Yaskawa INFORM job: apremTRJ5.JBI

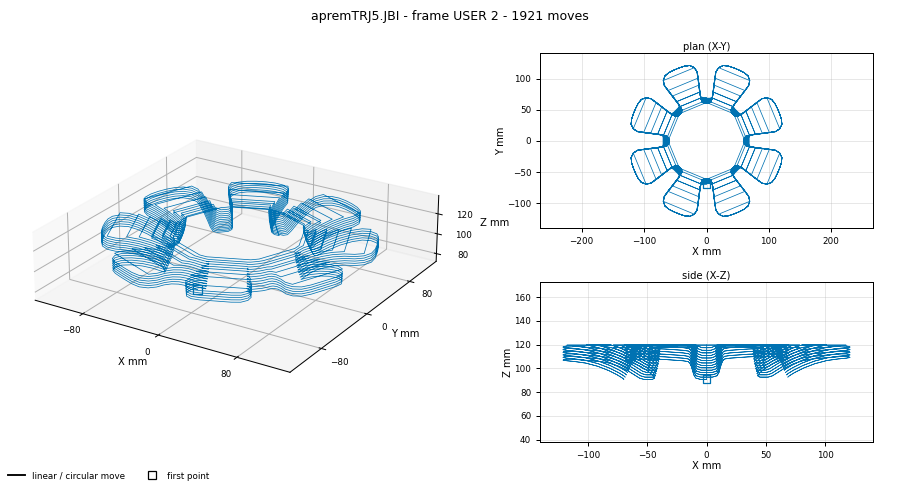
[picture p0: tool path of apremTRJ5.JBI in frame USER 2, 1921 of 1921 moves have a stored position in this frame; points joined in program order, loops and branches not executed]
/JOB
//NAME apremTRJ5
//POS
///NPOS 1921,0,0,0,0,0
///USER 2
///TOOL 1
///POSTYPE USER
///RECTAN
///RCONF 1,0,0,0,0,0,0,0,0,0,0,0,0,0,0,0,0,0,0,0,0,0,0,0
C00000=0.000,-69.663,90.662,149.0780,-0.0009,0.0000
C00001=-2.183,-69.638,90.631,149.0847,1.2932,0.0000
C00002=-5.231,-69.586,90.677,150.1957,-3.8236,0.0000
C00003=-9.064,-70.790,91.747,167.8852,-12.3668,0.0000
C00004=-10.724,-75.112,94.426,-179.6229,2.0642,0.0000
C00005=-11.710,-82.323,98.064,-179.4233,3.7476,0.0000
C00006=-12.828,-91.647,101.694,-179.3835,4.2590,0.0000
C00007=-14.066,-101.744,104.371,-179.3534,4.5111,0.0000
C00008=-15.480,-110.874,105.656,-178.6624,4.1341,0.0000
C00009=-19.937,-117.532,106.324,-177.9032,1.7507,0.0000
C00010=-26.978,-120.778,106.862,-178.7148,0.2137,0.0000
C00011=-35.142,-119.948,107.400,-179.9184,-0.0238,0.0000
C00012=-43.596,-117.150,107.753,-179.9908,-0.0034,0.0000
C00013=-52.010,-113.665,107.753,-179.9911,-0.0041,0.0000
C00014=-59.968,-109.665,107.400,-179.9255,-0.0409,0.0000
C00015=-66.327,-104.479,106.862,-179.2422,-1.0599,0.0000
C00016=-69.010,-97.206,106.324,-179.7550,-2.7196,0.0000
C00017=-67.454,-89.346,105.656,178.0185,-3.8685,0.0000
C00018=-61.998,-81.890,104.371,177.2629,-3.6488,0.0000
C00019=-55.734,-73.875,101.694,177.4206,-3.4489,0.0000
C00020=-49.931,-66.491,98.064,177.7552,-3.0586,0.0000
C00021=-45.529,-60.695,94.426,178.8066,-1.7264,0.0000
C00022=-43.647,-56.466,91.747,-179.8138,17.0577,0.0000
C00023=-45.506,-52.903,90.677,160.3117,24.3360,0.0000
C00024=-47.697,-50.786,90.631,156.2793,22.1709,0.0000
C00025=-49.259,-49.259,90.662,157.0437,22.9552,0.0000
C00026=-50.785,-47.698,90.631,157.8297,23.7213,0.0000
C00027=-52.904,-45.506,90.677,155.6631,19.6860,0.0000
C00028=-56.466,-43.647,91.747,162.9430,-0.1866,0.0000
C00029=-60.695,-45.529,94.426,-178.2736,1.1934,0.0000
C00030=-66.491,-49.931,98.064,-176.9414,2.2448,0.0000
C00031=-73.875,-55.734,101.694,-176.5511,2.5794,0.0000
C00032=-81.890,-61.998,104.371,-176.3512,2.7371,0.0000
C00033=-89.346,-67.454,105.656,-176.1315,1.9815,0.0000
C00034=-97.206,-69.010,106.324,-177.2804,-0.2450,0.0000
C00035=-104.479,-66.327,106.862,-178.9401,-0.7578,0.0000
C00036=-109.665,-59.968,107.400,-179.9591,-0.0745,0.0000
C00037=-113.665,-52.010,107.753,-179.9959,-0.0089,0.0000
C00038=-117.150,-43.596,107.753,-179.9966,-0.0092,0.0000
C00039=-119.948,-35.142,107.400,-179.9762,-0.0816,0.0000
C00040=-120.778,-26.978,106.862,179.7863,-1.2852,0.0000
C00041=-117.532,-19.937,106.324,178.2493,-2.0968,0.0000
C00042=-110.874,-15.480,105.656,175.8659,-1.3376,0.0000
C00043=-101.744,-14.066,104.371,175.4889,-0.6466,0.0000
C00044=-91.647,-12.828,101.694,175.7410,-0.6165,0.0000
C00045=-82.323,-11.710,98.064,176.2524,-0.5767,0.0000
C00046=-75.112,-10.724,94.426,177.9358,-0.3771,0.0000
C00047=-70.790,-9.064,91.747,-167.6330,12.1155,0.0000
C00048=-69.586,-5.231,90.677,-176.1790,29.8051,0.0000
C00049=-69.638,-2.184,90.631,178.7078,30.9153,0.0000
C00050=-69.663,0.000,90.662,179.9991,30.9220,0.0000
C00051=-69.638,2.183,90.631,-178.7068,30.9153,0.0000
C00052=-69.586,5.231,90.677,176.1764,29.8043,0.0000
C00053=-70.790,9.064,91.747,167.6332,12.1148,0.0000
C00054=-75.112,10.724,94.426,-177.9358,-0.3771,0.0000
C00055=-82.323,11.710,98.064,-176.2524,-0.5767,0.0000
C00056=-91.647,12.828,101.694,-175.7410,-0.6165,0.0000
C00057=-101.744,14.066,104.371,-175.4889,-0.6466,0.0000
C00058=-110.874,15.480,105.656,-175.8659,-1.3376,0.0000
C00059=-117.532,19.937,106.324,-178.2493,-2.0968,0.0000
C00060=-120.778,26.978,106.862,-179.7863,-1.2852,0.0000
C00061=-119.948,35.142,107.400,179.9762,-0.0816,0.0000
C00062=-117.150,43.596,107.753,179.9966,-0.0092,0.0000
C00063=-113.665,52.010,107.753,179.9959,-0.0089,0.0000
C00064=-109.665,59.968,107.400,179.9591,-0.0745,0.0000
C00065=-104.479,66.327,106.862,178.9401,-0.7578,0.0000
C00066=-97.206,69.010,106.324,177.2804,-0.2450,0.0000
C00067=-89.346,67.454,105.656,176.1315,1.9815,0.0000
C00068=-81.890,61.998,104.371,176.3512,2.7371,0.0000
C00069=-73.875,55.734,101.694,176.5511,2.5794,0.0000
C00070=-66.491,49.931,98.064,176.9414,2.2448,0.0000
C00071=-60.695,45.529,94.426,178.2736,1.1934,0.0000
C00072=-56.466,43.647,91.747,-162.9423,-0.1862,0.0000
C00073=-52.903,45.506,90.677,-155.6640,19.6883,0.0000
C00074=-50.786,47.697,90.631,-157.8291,23.7207,0.0000
C00075=-49.259,49.259,90.662,-157.0448,22.9563,0.0000
C00076=-47.698,50.785,90.631,-156.2787,22.1703,0.0000
C00077=-45.506,52.904,90.677,-160.3140,24.3369,0.0000
C00078=-43.647,56.466,91.747,179.8134,17.0570,0.0000
C00079=-45.529,60.695,94.426,-178.8066,-1.7264,0.0000
C00080=-49.931,66.491,98.064,-177.7552,-3.0586,0.0000
C00081=-55.734,73.875,101.694,-177.4206,-3.4489,0.0000
C00082=-61.998,81.890,104.371,-177.2629,-3.6488,0.0000
C00083=-67.454,89.346,105.656,-178.0185,-3.8685,0.0000
C00084=-69.010,97.206,106.324,179.7550,-2.7196,0.0000
C00085=-66.327,104.479,106.862,179.2422,-1.0599,0.0000
C00086=-59.968,109.665,107.400,179.9255,-0.0409,0.0000
C00087=-52.010,113.665,107.753,179.9911,-0.0041,0.0000
C00088=-43.596,117.150,107.753,179.9908,-0.0034,0.0000
C00089=-35.142,119.948,107.400,179.9184,-0.0238,0.0000
C00090=-26.978,120.778,106.862,178.7148,0.2137,0.0000
C00091=-19.937,117.532,106.324,177.9032,1.7507,0.0000
C00092=-15.480,110.874,105.656,178.6624,4.1341,0.0000
C00093=-14.066,101.744,104.371,179.3534,4.5111,0.0000
C00094=-12.828,91.647,101.694,179.3835,4.2590,0.0000
C00095=-11.710,82.323,98.064,179.4233,3.7476,0.0000
C00096=-10.724,75.112,94.426,179.6229,2.0642,0.0000
C00097=-9.064,70.790,91.747,-167.8852,-12.3668,0.0000
C00098=-5.231,69.586,90.677,-150.1957,-3.8236,0.0000
C00099=-2.183,69.638,90.631,-149.0847,1.2932,0.0000
C00100=0.000,69.663,90.662,-149.0780,-0.0009,0.0000
C00101=0.000,68.551,92.561,-150.2599,-0.0009,0.0000
C00102=2.082,68.530,92.529,-150.2645,-1.1898,0.0000
C00103=5.060,68.488,92.576,-151.4241,3.8705,0.0000
C00104=8.860,69.756,93.678,-168.9161,11.6642,0.0000
C00105=10.491,74.235,96.430,179.6271,-2.1340,0.0000
C00106=11.475,81.669,100.151,179.4707,-3.5332,0.0000
C00107=12.611,91.225,103.842,179.4509,-3.8705,0.0000
C00108=13.867,101.508,106.549,179.4410,-3.9839,0.0000
C00109=15.282,110.767,107.845,178.8532,-3.5972,0.0000
C00110=19.760,117.511,108.516,178.1979,-1.5173,0.0000
C00111=26.844,120.803,109.057,178.9013,-0.1852,0.0000
C00112=35.060,119.975,109.599,179.9308,0.0202,0.0000
C00113=43.570,117.160,109.952,179.9923,0.0029,0.0000
C00114=52.036,113.653,109.952,179.9925,0.0034,0.0000
C00115=60.044,109.627,109.599,179.9368,0.0347,0.0000
C00116=66.439,104.402,109.057,179.3540,0.9079,0.0000
C00117=69.120,97.065,108.516,179.7984,2.3465,0.0000
C00118=67.518,89.130,107.845,-178.2646,3.3542,0.0000
C00119=61.971,81.582,106.549,-177.5751,3.2135,0.0000
C00120=55.588,73.423,103.842,-177.6486,3.1262,0.0000
C00121=49.635,65.863,100.151,-177.8737,2.8734,0.0000
C00122=45.074,59.911,96.430,-178.7542,1.7728,0.0000
C00123=43.060,55.590,93.678,179.5731,-15.8809,0.0000
C00124=44.851,52.006,92.576,-161.3607,-23.4117,0.0000
C00125=46.985,49.930,92.529,-157.2861,-21.2671,0.0000
C00126=48.473,48.473,92.561,-158.0016,-21.9974,0.0000
C00127=49.930,46.986,92.529,-158.7334,-22.7144,0.0000
C00128=52.007,44.850,92.576,-156.5875,-18.6369,0.0000
C00129=55.590,43.060,93.678,-164.1198,0.4273,0.0000
C00130=59.911,45.074,96.430,178.2272,-1.2458,0.0000
C00131=65.863,49.635,100.151,177.1266,-2.1263,0.0000
C00132=73.423,55.588,103.842,176.8738,-2.3514,0.0000
C00133=81.582,61.971,106.549,176.7865,-2.4249,0.0000
C00134=89.130,67.518,107.845,176.6458,-1.7354,0.0000
C00135=97.065,69.120,108.516,177.6535,0.2016,0.0000
C00136=104.402,66.439,109.057,179.0921,0.6460,0.0000
C00137=109.627,60.044,109.599,179.9653,0.0632,0.0000
C00138=113.653,52.036,109.952,179.9966,0.0075,0.0000
C00139=117.160,43.570,109.952,179.9971,0.0077,0.0000
C00140=119.975,35.060,109.599,179.9798,0.0692,0.0000
C00141=120.803,26.844,109.057,-179.8148,1.0987,0.0000
C00142=117.511,19.760,108.516,-178.4827,1.8021,0.0000
C00143=110.767,15.282,107.845,-176.4028,1.1468,0.0000
C00144=101.508,13.867,106.549,-176.0161,0.5590,0.0000
C00145=91.225,12.611,103.842,-176.1295,0.5491,0.0000
C00146=81.669,11.475,100.151,-176.4668,0.5293,0.0000
C00147=74.235,10.491,96.430,-177.8660,0.3729,0.0000
C00148=69.756,8.860,93.678,168.3358,-11.0839,0.0000
C00149=68.488,5.060,92.576,176.1295,-28.5759,0.0000
C00150=68.530,2.082,92.529,-178.8102,-29.7355,0.0000
C00151=68.551,0.000,92.561,-179.9991,-29.7401,0.0000
C00152=68.530,-2.082,92.529,178.8093,-29.7356,0.0000
C00153=68.489,-5.060,92.576,-176.1270,-28.5749,0.0000
C00154=69.756,-8.860,93.678,-168.3360,-11.0832,0.0000
C00155=74.235,-10.491,96.430,177.8660,0.3729,0.0000
C00156=81.669,-11.475,100.151,176.4668,0.5293,0.0000
C00157=91.225,-12.611,103.842,176.1295,0.5491,0.0000
C00158=101.508,-13.867,106.549,176.0161,0.5590,0.0000
C00159=110.767,-15.282,107.845,176.4028,1.1468,0.0000
C00160=117.511,-19.760,108.516,178.4827,1.8021,0.0000
C00161=120.803,-26.844,109.057,179.8148,1.0987,0.0000
C00162=119.975,-35.060,109.599,-179.9798,0.0692,0.0000
C00163=117.160,-43.570,109.952,-179.9971,0.0077,0.0000
C00164=113.653,-52.036,109.952,-179.9966,0.0075,0.0000
C00165=109.627,-60.044,109.599,-179.9653,0.0632,0.0000
C00166=104.402,-66.439,109.057,-179.0921,0.6460,0.0000
C00167=97.065,-69.120,108.516,-177.6535,0.2016,0.0000
C00168=89.130,-67.518,107.845,-176.6458,-1.7354,0.0000
C00169=81.582,-61.971,106.549,-176.7865,-2.4249,0.0000
C00170=73.423,-55.588,103.842,-176.8738,-2.3514,0.0000
C00171=65.863,-49.635,100.151,-177.1266,-2.1263,0.0000
C00172=59.911,-45.074,96.430,-178.2272,-1.2458,0.0000
C00173=55.590,-43.060,93.678,164.1191,0.4269,0.0000
C00174=52.006,-44.851,92.576,156.5883,-18.6393,0.0000
C00175=49.930,-46.985,92.529,158.7329,-22.7139,0.0000
C00176=48.473,-48.473,92.561,158.0026,-21.9984,0.0000
C00177=46.986,-49.930,92.529,157.2856,-21.2666,0.0000
C00178=44.850,-52.007,92.576,161.3631,-23.4125,0.0000
C00179=43.060,-55.590,93.678,-179.5727,-15.8802,0.0000
C00180=45.074,-59.911,96.430,178.7542,1.7728,0.0000
C00181=49.635,-65.863,100.151,177.8737,2.8734,0.0000
C00182=55.588,-73.423,103.842,177.6486,3.1262,0.0000
C00183=61.971,-81.582,106.549,177.5751,3.2135,0.0000
C00184=67.518,-89.130,107.845,178.2646,3.3542,0.0000
C00185=69.120,-97.065,108.516,-179.7984,2.3465,0.0000
C00186=66.439,-104.402,109.057,-179.3540,0.9079,0.0000
C00187=60.044,-109.627,109.599,-179.9368,0.0347,0.0000
C00188=52.036,-113.653,109.952,-179.9925,0.0034,0.0000
C00189=43.570,-117.160,109.952,-179.9923,0.0029,0.0000
C00190=35.060,-119.975,109.599,-179.9308,0.0202,0.0000
C00191=26.844,-120.803,109.057,-178.9013,-0.1852,0.0000
C00192=19.760,-117.511,108.516,-178.1979,-1.5173,0.0000
C00193=15.282,-110.767,107.845,-178.8532,-3.5972,0.0000
C00194=13.867,-101.508,106.549,-179.4410,-3.9839,0.0000
C00195=12.611,-91.225,103.842,-179.4509,-3.8705,0.0000
C00196=11.475,-81.669,100.151,-179.4707,-3.5332,0.0000
C00197=10.491,-74.235,96.430,-179.6271,-2.1340,0.0000
C00198=8.860,-69.756,93.678,168.9161,11.6642,0.0000
C00199=5.060,-68.488,92.576,151.4241,3.8705,0.0000
C00200=2.082,-68.530,92.529,150.2645,-1.1898,0.0000
C00201=0.000,-68.551,92.561,150.2599,-0.0009,0.0000
C00202=0.000,-68.551,92.561,150.2599,-0.0009,0.0000
C00203=-2.082,-68.530,92.529,150.2644,1.1907,0.0000
C00204=-5.060,-68.489,92.576,151.4251,-3.8730,0.0000
C00205=-8.860,-69.756,93.678,168.9168,-11.6640,0.0000
C00206=-10.491,-74.235,96.430,-179.6271,2.1340,0.0000
C00207=-11.475,-81.669,100.151,-179.4707,3.5332,0.0000
C00208=-12.611,-91.225,103.842,-179.4509,3.8705,0.0000
C00209=-13.867,-101.508,106.549,-179.4410,3.9839,0.0000
C00210=-15.282,-110.767,107.845,-178.8532,3.5972,0.0000
C00211=-19.760,-117.511,108.516,-178.1979,1.5173,0.0000
C00212=-26.844,-120.803,109.057,-178.9013,0.1852,0.0000
C00213=-35.060,-119.975,109.599,-179.9308,-0.0202,0.0000
C00214=-43.570,-117.160,109.952,-179.9923,-0.0029,0.0000
C00215=-52.036,-113.653,109.952,-179.9925,-0.0034,0.0000
C00216=-60.044,-109.627,109.599,-179.9368,-0.0347,0.0000
C00217=-66.439,-104.402,109.057,-179.3540,-0.9079,0.0000
C00218=-69.120,-97.065,108.516,-179.7984,-2.3465,0.0000
C00219=-67.518,-89.130,107.845,178.2646,-3.3542,0.0000
C00220=-61.971,-81.582,106.549,177.5751,-3.2135,0.0000
C00221=-55.588,-73.423,103.842,177.6486,-3.1262,0.0000
C00222=-49.635,-65.863,100.151,177.8737,-2.8734,0.0000
C00223=-45.074,-59.911,96.430,178.7542,-1.7728,0.0000
C00224=-43.060,-55.590,93.678,-179.5731,15.8809,0.0000
C00225=-44.851,-52.006,92.576,161.3607,23.4117,0.0000
C00226=-46.985,-49.930,92.529,157.2861,21.2671,0.0000
C00227=-48.473,-48.473,92.561,158.0016,21.9974,0.0000
C00228=-49.930,-46.986,92.529,158.7334,22.7144,0.0000
C00229=-52.007,-44.850,92.576,156.5875,18.6369,0.0000
C00230=-55.590,-43.060,93.678,164.1198,-0.4273,0.0000
C00231=-59.911,-45.074,96.430,-178.2272,1.2458,0.0000
C00232=-65.863,-49.635,100.151,-177.1266,2.1263,0.0000
C00233=-73.423,-55.588,103.842,-176.8738,2.3514,0.0000
C00234=-81.582,-61.971,106.549,-176.7865,2.4249,0.0000
C00235=-89.130,-67.518,107.845,-176.6458,1.7354,0.0000
C00236=-97.065,-69.120,108.516,-177.6535,-0.2016,0.0000
C00237=-104.402,-66.439,109.057,-179.0921,-0.6460,0.0000
C00238=-109.627,-60.044,109.599,-179.9653,-0.0632,0.0000
C00239=-113.653,-52.036,109.952,-179.9966,-0.0075,0.0000
C00240=-117.160,-43.570,109.952,-179.9971,-0.0077,0.0000
C00241=-119.975,-35.060,109.599,-179.9798,-0.0692,0.0000
C00242=-120.803,-26.844,109.057,179.8148,-1.0987,0.0000
C00243=-117.511,-19.760,108.516,178.4827,-1.8021,0.0000
C00244=-110.767,-15.282,107.845,176.4028,-1.1468,0.0000
C00245=-101.508,-13.867,106.549,176.0161,-0.5590,0.0000
C00246=-91.225,-12.611,103.842,176.1295,-0.5491,0.0000
C00247=-81.669,-11.475,100.151,176.4668,-0.5293,0.0000
C00248=-74.235,-10.491,96.430,177.8660,-0.3729,0.0000
C00249=-69.756,-8.860,93.678,-168.3358,11.0839,0.0000
C00250=-68.488,-5.060,92.576,-176.1295,28.5759,0.0000
C00251=-68.530,-2.082,92.529,178.8102,29.7355,0.0000
C00252=-68.551,0.000,92.561,179.9991,29.7401,0.0000
C00253=-68.530,2.082,92.529,-178.8093,29.7356,0.0000
C00254=-68.489,5.060,92.576,176.1270,28.5749,0.0000
C00255=-69.756,8.860,93.678,168.3360,11.0832,0.0000
C00256=-74.235,10.491,96.430,-177.8660,-0.3729,0.0000
C00257=-81.669,11.475,100.151,-176.4668,-0.5293,0.0000
C00258=-91.225,12.611,103.842,-176.1295,-0.5491,0.0000
C00259=-101.508,13.867,106.549,-176.0161,-0.5590,0.0000
C00260=-110.767,15.282,107.845,-176.4028,-1.1468,0.0000
C00261=-117.511,19.760,108.516,-178.4827,-1.8021,0.0000
C00262=-120.803,26.844,109.057,-179.8148,-1.0987,0.0000
C00263=-119.975,35.060,109.599,179.9798,-0.0692,0.0000
C00264=-117.160,43.570,109.952,179.9971,-0.0077,0.0000
C00265=-113.653,52.036,109.952,179.9966,-0.0075,0.0000
C00266=-109.627,60.044,109.599,179.9653,-0.0632,0.0000
C00267=-104.402,66.439,109.057,179.0921,-0.6460,0.0000
C00268=-97.065,69.120,108.516,177.6535,-0.2016,0.0000
C00269=-89.130,67.518,107.845,176.6458,1.7354,0.0000
C00270=-81.582,61.971,106.549,176.7865,2.4249,0.0000
C00271=-73.423,55.588,103.842,176.8738,2.3514,0.0000
C00272=-65.863,49.635,100.151,177.1266,2.1263,0.0000
C00273=-59.911,45.074,96.430,178.2272,1.2458,0.0000
C00274=-55.590,43.060,93.678,-164.1191,-0.4269,0.0000
C00275=-52.006,44.851,92.576,-156.5883,18.6393,0.0000
C00276=-49.930,46.985,92.529,-158.7329,22.7139,0.0000
C00277=-48.473,48.473,92.561,-158.0026,21.9984,0.0000
C00278=-46.986,49.930,92.529,-157.2856,21.2666,0.0000
C00279=-44.850,52.007,92.576,-161.3631,23.4125,0.0000
C00280=-43.060,55.590,93.678,179.5727,15.8802,0.0000
C00281=-45.074,59.911,96.430,-178.7542,-1.7728,0.0000
C00282=-49.635,65.863,100.151,-177.8737,-2.8734,0.0000
C00283=-55.588,73.423,103.842,-177.6486,-3.1262,0.0000
C00284=-61.971,81.582,106.549,-177.5751,-3.2135,0.0000
C00285=-67.518,89.130,107.845,-178.2646,-3.3542,0.0000
C00286=-69.120,97.065,108.516,179.7984,-2.3465,0.0000
C00287=-66.439,104.402,109.057,179.3540,-0.9079,0.0000
C00288=-60.044,109.627,109.599,179.9368,-0.0347,0.0000
C00289=-52.036,113.653,109.952,179.9925,-0.0034,0.0000
C00290=-43.570,117.160,109.952,179.9923,-0.0029,0.0000
C00291=-35.060,119.975,109.599,179.9308,-0.0202,0.0000
C00292=-26.844,120.803,109.057,178.9013,0.1852,0.0000
C00293=-19.760,117.511,108.516,178.1979,1.5173,0.0000
C00294=-15.282,110.767,107.845,178.8532,3.5972,0.0000
C00295=-13.867,101.508,106.549,179.4410,3.9839,0.0000
C00296=-12.611,91.225,103.842,179.4509,3.8705,0.0000
C00297=-11.475,81.669,100.151,179.4707,3.5332,0.0000
C00298=-10.491,74.235,96.430,179.6271,2.1340,0.0000
C00299=-8.860,69.756,93.678,-168.9168,-11.6640,0.0000
C00300=-5.060,68.489,92.576,-151.4251,-3.8730,0.0000
C00301=-2.082,68.530,92.529,-150.2644,1.1907,0.0000
C00302=0.000,68.551,92.561,-150.2599,-0.0009,0.0000
C00303=0.000,67.481,94.483,-151.5573,-0.0008,0.0000
C00304=1.984,67.463,94.450,-151.5596,-1.0856,0.0000
C00305=4.895,67.432,94.499,-152.7618,3.8795,0.0000
C00306=8.665,68.764,95.632,-169.9184,10.9214,0.0000
C00307=10.271,73.406,98.456,179.6393,-2.1542,0.0000
C00308=11.257,81.064,102.255,179.5203,-3.2821,0.0000
C00309=12.417,90.845,106.000,179.5197,-3.4475,0.0000
C00310=13.694,101.302,108.733,179.5288,-3.4203,0.0000
C00311=15.114,110.675,110.036,179.0481,-3.0234,0.0000
C00312=19.611,117.493,110.711,178.5095,-1.2637,0.0000
C00313=26.731,120.823,111.254,179.1000,-0.1534,0.0000
C00314=34.993,119.997,111.797,179.9440,0.0163,0.0000
C00315=43.548,117.168,112.152,179.9938,0.0023,0.0000
C00316=52.058,113.643,112.152,179.9940,0.0028,0.0000
C00317=60.107,109.595,111.797,179.9489,0.0281,0.0000
C00318=66.533,104.337,111.254,179.4720,0.7449,0.0000
C00319=69.213,96.947,110.711,179.8395,1.9472,0.0000
C00320=67.572,88.946,110.036,-178.5336,2.8107,0.0000
C00321=61.948,81.315,108.733,-177.9127,2.7525,0.0000
C00322=55.457,73.018,106.000,-177.8999,2.7782,0.0000
C00323=49.361,65.281,102.255,-178.0167,2.6606,0.0000
C00324=44.643,59.169,98.456,-178.7313,1.7785,0.0000
C00325=42.497,54.751,95.632,179.3858,-14.6902,0.0000
C00326=44.220,51.143,94.499,-162.4610,-22.3893,0.0000
C00327=46.300,49.106,94.450,-158.3778,-20.2832,0.0000
C00328=47.716,47.716,94.483,-159.0421,-20.9569,0.0000
C00329=49.106,46.300,94.450,-159.7173,-21.6227,0.0000
C00330=51.144,44.220,94.499,-157.6099,-17.5367,0.0000
C00331=54.751,42.497,95.632,-165.3105,0.6146,0.0000
C00332=59.169,44.643,98.456,178.2215,-1.2687,0.0000
C00333=65.281,49.361,102.255,177.3394,-1.9833,0.0000
C00334=73.018,55.457,106.000,177.2218,-2.1001,0.0000
C00335=81.315,61.948,108.733,177.2475,-2.0873,0.0000
C00336=88.946,67.572,110.036,177.1893,-1.4664,0.0000
C00337=96.947,69.213,110.711,178.0528,0.1605,0.0000
C00338=104.337,66.533,111.254,179.2551,0.5280,0.0000
C00339=109.595,60.107,111.797,179.9719,0.0511,0.0000
C00340=113.643,52.058,112.152,179.9972,0.0060,0.0000
C00341=117.168,43.548,112.152,179.9977,0.0062,0.0000
C00342=119.997,34.993,111.797,179.9837,0.0560,0.0000
C00343=120.823,26.731,111.254,-179.8466,0.9000,0.0000
C00344=117.493,19.611,110.711,-178.7363,1.4905,0.0000
C00345=110.675,15.114,110.036,-176.9766,0.9519,0.0000
C00346=101.302,13.694,108.733,-176.5797,0.4712,0.0000
C00347=90.845,12.417,106.000,-176.5525,0.4803,0.0000
C00348=81.064,11.257,102.255,-176.7179,0.4797,0.0000
C00349=73.406,10.271,98.456,-177.8458,0.3607,0.0000
C00350=68.764,8.665,95.632,169.0786,-10.0816,0.0000
C00351=67.432,4.895,94.499,176.1205,-27.2382,0.0000
C00352=67.463,1.984,94.450,-178.9144,-28.4404,0.0000
C00353=67.481,0.000,94.483,-179.9992,-28.4427,0.0000
C00354=67.463,-1.984,94.450,178.9136,-28.4404,0.0000
C00355=67.432,-4.896,94.499,-176.1180,-27.2373,0.0000
C00356=68.764,-8.665,95.632,-169.0788,-10.0808,0.0000
C00357=73.406,-10.271,98.456,177.8458,0.3607,0.0000
C00358=81.064,-11.257,102.255,176.7179,0.4797,0.0000
C00359=90.845,-12.417,106.000,176.5525,0.4803,0.0000
C00360=101.302,-13.694,108.733,176.5797,0.4712,0.0000
C00361=110.675,-15.114,110.036,176.9766,0.9519,0.0000
C00362=117.493,-19.611,110.711,178.7363,1.4905,0.0000
C00363=120.823,-26.731,111.254,179.8466,0.9000,0.0000
C00364=119.997,-34.993,111.797,-179.9837,0.0560,0.0000
C00365=117.168,-43.548,112.152,-179.9977,0.0062,0.0000
C00366=113.643,-52.058,112.152,-179.9972,0.0060,0.0000
C00367=109.595,-60.107,111.797,-179.9719,0.0511,0.0000
C00368=104.337,-66.533,111.254,-179.2551,0.5280,0.0000
C00369=96.947,-69.213,110.711,-178.0528,0.1605,0.0000
C00370=88.946,-67.572,110.036,-177.1893,-1.4664,0.0000
C00371=81.315,-61.948,108.733,-177.2475,-2.0873,0.0000
C00372=73.018,-55.457,106.000,-177.2218,-2.1001,0.0000
C00373=65.281,-49.361,102.255,-177.3394,-1.9833,0.0000
C00374=59.169,-44.643,98.456,-178.2215,-1.2687,0.0000
C00375=54.751,-42.497,95.632,165.3098,0.6142,0.0000
C00376=51.143,-44.220,94.499,157.6107,-17.5390,0.0000
C00377=49.106,-46.300,94.450,159.7168,-21.6222,0.0000
C00378=47.716,-47.716,94.483,159.0431,-20.9579,0.0000
C00379=46.300,-49.106,94.450,158.3773,-20.2827,0.0000
C00380=44.220,-51.144,94.499,162.4633,-22.3901,0.0000
C00381=42.497,-54.751,95.632,-179.3854,-14.6895,0.0000
C00382=44.643,-59.169,98.456,178.7313,1.7785,0.0000
C00383=49.361,-65.281,102.255,178.0167,2.6606,0.0000
C00384=55.457,-73.018,106.000,177.8999,2.7782,0.0000
C00385=61.948,-81.315,108.733,177.9127,2.7525,0.0000
C00386=67.572,-88.946,110.036,178.5336,2.8107,0.0000
C00387=69.213,-96.947,110.711,-179.8395,1.9472,0.0000
C00388=66.533,-104.337,111.254,-179.4720,0.7449,0.0000
C00389=60.107,-109.595,111.797,-179.9489,0.0281,0.0000
C00390=52.058,-113.643,112.152,-179.9940,0.0028,0.0000
C00391=43.548,-117.168,112.152,-179.9938,0.0023,0.0000
C00392=34.993,-119.997,111.797,-179.9440,0.0163,0.0000
C00393=26.731,-120.823,111.254,-179.1000,-0.1534,0.0000
C00394=19.611,-117.493,110.711,-178.5095,-1.2637,0.0000
C00395=15.114,-110.675,110.036,-179.0481,-3.0234,0.0000
C00396=13.694,-101.302,108.733,-179.5288,-3.4203,0.0000
C00397=12.417,-90.845,106.000,-179.5197,-3.4475,0.0000
C00398=11.257,-81.064,102.255,-179.5203,-3.2821,0.0000
C00399=10.271,-73.406,98.456,-179.6393,-2.1542,0.0000
C00400=8.665,-68.764,95.632,169.9184,10.9214,0.0000
C00401=4.895,-67.432,94.499,152.7618,3.8795,0.0000
C00402=1.984,-67.463,94.450,151.5596,-1.0856,0.0000
C00403=0.000,-67.481,94.483,151.5573,-0.0008,0.0000
C00404=0.000,-67.481,94.483,151.5573,-0.0008,0.0000
C00405=-1.984,-67.463,94.450,151.5596,1.0864,0.0000
C00406=-4.896,-67.432,94.499,152.7627,-3.8820,0.0000
C00407=-8.665,-68.764,95.632,169.9192,-10.9212,0.0000
C00408=-10.271,-73.406,98.456,-179.6393,2.1542,0.0000
C00409=-11.257,-81.064,102.255,-179.5203,3.2821,0.0000
C00410=-12.417,-90.845,106.000,-179.5197,3.4475,0.0000
C00411=-13.694,-101.302,108.733,-179.5288,3.4203,0.0000
C00412=-15.114,-110.675,110.036,-179.0481,3.0234,0.0000
C00413=-19.611,-117.493,110.711,-178.5095,1.2637,0.0000
C00414=-26.731,-120.823,111.254,-179.1000,0.1534,0.0000
C00415=-34.993,-119.997,111.797,-179.9440,-0.0163,0.0000
C00416=-43.548,-117.168,112.152,-179.9938,-0.0023,0.0000
C00417=-52.058,-113.643,112.152,-179.9940,-0.0028,0.0000
C00418=-60.107,-109.595,111.797,-179.9489,-0.0281,0.0000
C00419=-66.533,-104.337,111.254,-179.4720,-0.7449,0.0000
C00420=-69.213,-96.947,110.711,-179.8395,-1.9472,0.0000
C00421=-67.572,-88.946,110.036,178.5336,-2.8107,0.0000
C00422=-61.948,-81.315,108.733,177.9127,-2.7525,0.0000
C00423=-55.457,-73.018,106.000,177.8999,-2.7782,0.0000
C00424=-49.361,-65.281,102.255,178.0167,-2.6606,0.0000
C00425=-44.643,-59.169,98.456,178.7313,-1.7785,0.0000
C00426=-42.497,-54.751,95.632,-179.3858,14.6902,0.0000
C00427=-44.220,-51.143,94.499,162.4610,22.3893,0.0000
C00428=-46.300,-49.106,94.450,158.3778,20.2832,0.0000
C00429=-47.716,-47.716,94.483,159.0421,20.9569,0.0000
C00430=-49.106,-46.300,94.450,159.7173,21.6227,0.0000
C00431=-51.144,-44.220,94.499,157.6099,17.5367,0.0000
C00432=-54.751,-42.497,95.632,165.3105,-0.6146,0.0000
C00433=-59.169,-44.643,98.456,-178.2215,1.2687,0.0000
C00434=-65.281,-49.361,102.255,-177.3394,1.9833,0.0000
C00435=-73.018,-55.457,106.000,-177.2218,2.1001,0.0000
C00436=-81.315,-61.948,108.733,-177.2475,2.0873,0.0000
C00437=-88.946,-67.572,110.036,-177.1893,1.4664,0.0000
C00438=-96.947,-69.213,110.711,-178.0528,-0.1605,0.0000
C00439=-104.337,-66.533,111.254,-179.2551,-0.5280,0.0000
C00440=-109.595,-60.107,111.797,-179.9719,-0.0511,0.0000
C00441=-113.643,-52.058,112.152,-179.9972,-0.0060,0.0000
C00442=-117.168,-43.548,112.152,-179.9977,-0.0062,0.0000
C00443=-119.997,-34.993,111.797,-179.9837,-0.0560,0.0000
C00444=-120.823,-26.731,111.254,179.8466,-0.9000,0.0000
C00445=-117.493,-19.611,110.711,178.7363,-1.4905,0.0000
C00446=-110.675,-15.114,110.036,176.9766,-0.9519,0.0000
C00447=-101.302,-13.694,108.733,176.5797,-0.4712,0.0000
C00448=-90.845,-12.417,106.000,176.5525,-0.4803,0.0000
C00449=-81.064,-11.257,102.255,176.7179,-0.4797,0.0000
C00450=-73.406,-10.271,98.456,177.8458,-0.3607,0.0000
C00451=-68.764,-8.665,95.632,-169.0786,10.0816,0.0000
C00452=-67.432,-4.895,94.499,-176.1205,27.2382,0.0000
C00453=-67.463,-1.984,94.450,178.9144,28.4404,0.0000
C00454=-67.481,0.000,94.483,179.9992,28.4427,0.0000
C00455=-67.463,1.984,94.450,-178.9136,28.4404,0.0000
C00456=-67.432,4.896,94.499,176.1180,27.2373,0.0000
C00457=-68.764,8.665,95.632,169.0788,10.0808,0.0000
C00458=-73.406,10.271,98.456,-177.8458,-0.3607,0.0000
C00459=-81.064,11.257,102.255,-176.7179,-0.4797,0.0000
C00460=-90.845,12.417,106.000,-176.5525,-0.4803,0.0000
C00461=-101.302,13.694,108.733,-176.5797,-0.4712,0.0000
C00462=-110.675,15.114,110.036,-176.9766,-0.9519,0.0000
C00463=-117.493,19.611,110.711,-178.7363,-1.4905,0.0000
C00464=-120.823,26.731,111.254,-179.8466,-0.9000,0.0000
C00465=-119.997,34.993,111.797,179.9837,-0.0560,0.0000
C00466=-117.168,43.548,112.152,179.9977,-0.0062,0.0000
C00467=-113.643,52.058,112.152,179.9972,-0.0060,0.0000
C00468=-109.595,60.107,111.797,179.9719,-0.0511,0.0000
C00469=-104.337,66.533,111.254,179.2551,-0.5280,0.0000
C00470=-96.947,69.213,110.711,178.0528,-0.1605,0.0000
C00471=-88.946,67.572,110.036,177.1893,1.4664,0.0000
C00472=-81.315,61.948,108.733,177.2475,2.0873,0.0000
C00473=-73.018,55.457,106.000,177.2218,2.1001,0.0000
C00474=-65.281,49.361,102.255,177.3394,1.9833,0.0000
C00475=-59.169,44.643,98.456,178.2215,1.2687,0.0000
C00476=-54.751,42.497,95.632,-165.3098,-0.6142,0.0000
C00477=-51.143,44.220,94.499,-157.6107,17.5390,0.0000
C00478=-49.106,46.300,94.450,-159.7168,21.6222,0.0000
C00479=-47.716,47.716,94.483,-159.0431,20.9579,0.0000
C00480=-46.300,49.106,94.450,-158.3773,20.2827,0.0000
C00481=-44.220,51.144,94.499,-162.4633,22.3901,0.0000
C00482=-42.497,54.751,95.632,179.3854,14.6895,0.0000
C00483=-44.643,59.169,98.456,-178.7313,-1.7785,0.0000
C00484=-49.361,65.281,102.255,-178.0167,-2.6606,0.0000
C00485=-55.457,73.018,106.000,-177.8999,-2.7782,0.0000
C00486=-61.948,81.315,108.733,-177.9127,-2.7525,0.0000
C00487=-67.572,88.946,110.036,-178.5336,-2.8107,0.0000
C00488=-69.213,96.947,110.711,179.8395,-1.9472,0.0000
C00489=-66.533,104.337,111.254,179.4720,-0.7449,0.0000
C00490=-60.107,109.595,111.797,179.9489,-0.0281,0.0000
C00491=-52.058,113.643,112.152,179.9940,-0.0028,0.0000
C00492=-43.548,117.168,112.152,179.9938,-0.0023,0.0000
C00493=-34.993,119.997,111.797,179.9440,-0.0163,0.0000
C00494=-26.731,120.823,111.254,179.1000,0.1534,0.0000
C00495=-19.611,117.493,110.711,178.5095,1.2637,0.0000
C00496=-15.114,110.675,110.036,179.0481,3.0234,0.0000
C00497=-13.694,101.302,108.733,179.5288,3.4203,0.0000
C00498=-12.417,90.845,106.000,179.5197,3.4475,0.0000
C00499=-11.257,81.064,102.255,179.5203,3.2821,0.0000
C00500=-10.271,73.406,98.456,179.6393,2.1542,0.0000
C00501=-8.665,68.764,95.632,-169.9192,-10.9212,0.0000
C00502=-4.896,67.432,94.499,-152.7627,-3.8820,0.0000
C00503=-1.984,67.463,94.450,-151.5596,1.0864,0.0000
C00504=0.000,67.481,94.483,-151.5573,-0.0008,0.0000
C00505=0.000,66.457,96.430,-152.9799,-0.0007,0.0000
C00506=1.891,66.441,96.396,-152.9796,-0.9804,0.0000
C00507=4.738,66.421,96.447,-154.2147,3.8448,0.0000
C00508=8.479,67.820,97.611,-170.8911,10.1417,0.0000
C00509=10.065,72.628,100.503,179.6580,-2.1261,0.0000
C00510=11.059,80.512,104.375,179.5721,-2.9949,0.0000
C00511=12.247,90.513,108.168,179.5898,-2.9910,0.0000
C00512=13.549,101.129,110.921,179.6173,-2.8213,0.0000
C00513=14.976,110.600,112.231,179.2477,-2.4139,0.0000
C00514=19.491,117.478,112.908,178.8374,-0.9912,0.0000
C00515=26.642,120.839,113.453,179.3104,-0.1186,0.0000
C00516=34.941,120.015,113.997,179.9580,0.0122,0.0000
C00517=43.531,117.175,114.352,179.9954,0.0017,0.0000
C00518=52.074,113.636,114.352,179.9956,0.0020,0.0000
C00519=60.156,109.570,113.997,179.9617,0.0211,0.0000
C00520=66.607,104.285,113.453,179.5962,0.5715,0.0000
C00521=69.288,96.852,112.908,179.8787,1.5228,0.0000
C00522=67.616,88.795,112.231,-178.8242,2.2388,0.0000
C00523=61.928,81.090,110.921,-178.2745,2.2660,0.0000
C00524=55.342,72.662,108.168,-178.1738,2.4056,0.0000
C00525=49.111,64.751,104.375,-178.1836,2.4208,0.0000
C00526=44.239,58.473,100.503,-178.7380,1.7453,0.0000
C00527=41.961,53.951,97.611,179.2487,-13.4881,0.0000
C00528=43.616,50.317,96.447,-163.6122,-21.2623,0.0000
C00529=45.644,48.318,96.396,-159.5592,-19.2137,0.0000
C00530=46.992,46.992,96.430,-160.1702,-19.8289,0.0000
C00531=48.317,45.644,96.396,-160.7867,-20.4413,0.0000
C00532=50.318,43.616,96.447,-158.7369,-16.3854,0.0000
C00533=53.952,41.961,97.611,-166.5126,0.7516,0.0000
C00534=58.473,44.239,100.503,178.2547,-1.2620,0.0000
C00535=64.751,49.111,104.375,177.5792,-1.8164,0.0000
C00536=72.662,55.342,108.168,177.5944,-1.8262,0.0000
C00537=81.090,61.928,110.921,177.7340,-1.7255,0.0000
C00538=88.795,67.616,112.231,177.7612,-1.1758,0.0000
C00539=96.852,69.288,112.908,178.4772,0.1213,0.0000
C00540=104.285,66.607,113.453,179.4285,0.4038,0.0000
C00541=109.570,60.156,113.997,179.9789,0.0383,0.0000
C00542=113.636,52.074,114.352,179.9980,0.0044,0.0000
C00543=117.175,43.531,114.352,179.9983,0.0046,0.0000
C00544=120.015,34.941,113.997,179.9878,0.0420,0.0000
C00545=120.839,26.642,113.453,-179.8814,0.6896,0.0000
C00546=117.478,19.491,112.908,-179.0088,1.1626,0.0000
C00547=110.600,14.976,112.231,-177.5861,0.7523,0.0000
C00548=101.129,13.549,110.921,-177.1787,0.3827,0.0000
C00549=90.513,12.247,108.168,-177.0090,0.4102,0.0000
C00550=80.512,11.059,104.375,-177.0051,0.4279,0.0000
C00551=72.628,10.065,100.503,-177.8739,0.3420,0.0000
C00552=67.820,8.479,97.611,169.8583,-9.1089,0.0000
C00553=66.421,4.738,96.447,176.1552,-25.7853,0.0000
C00554=66.441,1.891,96.396,-179.0196,-27.0204,0.0000
C00555=66.457,0.000,96.430,-179.9993,-27.0201,0.0000
C00556=66.441,-1.890,96.396,179.0188,-27.0205,0.0000
C00557=66.421,-4.739,96.447,-176.1528,-25.7844,0.0000
C00558=67.820,-8.479,97.611,-169.8585,-9.1082,0.0000
C00559=72.628,-10.065,100.503,177.8739,0.3420,0.0000
C00560=80.512,-11.059,104.375,177.0051,0.4279,0.0000
C00561=90.513,-12.247,108.168,177.0090,0.4102,0.0000
C00562=101.129,-13.549,110.921,177.1787,0.3827,0.0000
C00563=110.600,-14.976,112.231,177.5861,0.7523,0.0000
C00564=117.478,-19.491,112.908,179.0088,1.1626,0.0000
C00565=120.839,-26.642,113.453,179.8814,0.6896,0.0000
C00566=120.015,-34.941,113.997,-179.9878,0.0420,0.0000
C00567=117.175,-43.531,114.352,-179.9983,0.0046,0.0000
C00568=113.636,-52.074,114.352,-179.9980,0.0044,0.0000
C00569=109.570,-60.156,113.997,-179.9789,0.0383,0.0000
C00570=104.285,-66.607,113.453,-179.4285,0.4038,0.0000
C00571=96.852,-69.288,112.908,-178.4772,0.1213,0.0000
C00572=88.795,-67.616,112.231,-177.7612,-1.1758,0.0000
C00573=81.090,-61.928,110.921,-177.7340,-1.7255,0.0000
C00574=72.662,-55.342,108.168,-177.5944,-1.8262,0.0000
C00575=64.751,-49.111,104.375,-177.5792,-1.8164,0.0000
C00576=58.473,-44.239,100.503,-178.2547,-1.2620,0.0000
C00577=53.951,-41.961,97.611,166.5119,0.7513,0.0000
C00578=50.317,-43.616,96.447,158.7377,-16.3878,0.0000
C00579=48.318,-45.644,96.396,160.7863,-20.4408,0.0000
C00580=46.992,-46.992,96.430,160.1711,-19.8298,0.0000
C00581=45.644,-48.317,96.396,159.5587,-19.2133,0.0000
C00582=43.616,-50.318,96.447,163.6146,-21.2631,0.0000
C00583=41.961,-53.952,97.611,-179.2484,-13.4874,0.0000
C00584=44.239,-58.473,100.503,178.7380,1.7453,0.0000
C00585=49.111,-64.751,104.375,178.1836,2.4208,0.0000
C00586=55.342,-72.662,108.168,178.1738,2.4056,0.0000
C00587=61.928,-81.090,110.921,178.2745,2.2660,0.0000
C00588=67.616,-88.795,112.231,178.8242,2.2388,0.0000
C00589=69.288,-96.852,112.908,-179.8787,1.5228,0.0000
C00590=66.607,-104.285,113.453,-179.5962,0.5715,0.0000
C00591=60.156,-109.570,113.997,-179.9617,0.0211,0.0000
C00592=52.074,-113.636,114.352,-179.9956,0.0020,0.0000
C00593=43.531,-117.175,114.352,-179.9954,0.0017,0.0000
C00594=34.941,-120.015,113.997,-179.9580,0.0122,0.0000
C00595=26.642,-120.839,113.453,-179.3104,-0.1186,0.0000
C00596=19.491,-117.478,112.908,-178.8374,-0.9912,0.0000
C00597=14.976,-110.600,112.231,-179.2477,-2.4139,0.0000
C00598=13.549,-101.129,110.921,-179.6173,-2.8213,0.0000
C00599=12.247,-90.513,108.168,-179.5898,-2.9910,0.0000
C00600=11.059,-80.512,104.375,-179.5721,-2.9949,0.0000
C00601=10.065,-72.628,100.503,-179.6580,-2.1261,0.0000
C00602=8.479,-67.820,97.611,170.8911,10.1417,0.0000
C00603=4.738,-66.421,96.447,154.2147,3.8448,0.0000
C00604=1.891,-66.441,96.396,152.9796,-0.9804,0.0000
C00605=0.000,-66.457,96.430,152.9799,-0.0007,0.0000
C00606=0.000,-66.457,96.430,152.9799,-0.0007,0.0000
C00607=-1.890,-66.441,96.396,152.9795,0.9812,0.0000
C00608=-4.739,-66.421,96.447,154.2156,-3.8472,0.0000
C00609=-8.479,-67.820,97.611,170.8918,-10.1415,0.0000
C00610=-10.065,-72.628,100.503,-179.6580,2.1261,0.0000
C00611=-11.059,-80.512,104.375,-179.5721,2.9949,0.0000
C00612=-12.247,-90.513,108.168,-179.5898,2.9910,0.0000
C00613=-13.549,-101.129,110.921,-179.6173,2.8213,0.0000
C00614=-14.976,-110.600,112.231,-179.2477,2.4139,0.0000
C00615=-19.491,-117.478,112.908,-178.8374,0.9912,0.0000
C00616=-26.642,-120.839,113.453,-179.3104,0.1186,0.0000
C00617=-34.941,-120.015,113.997,-179.9580,-0.0122,0.0000
C00618=-43.531,-117.175,114.352,-179.9954,-0.0017,0.0000
C00619=-52.074,-113.636,114.352,-179.9956,-0.0020,0.0000
C00620=-60.156,-109.570,113.997,-179.9617,-0.0211,0.0000
C00621=-66.607,-104.285,113.453,-179.5962,-0.5715,0.0000
C00622=-69.288,-96.852,112.908,-179.8787,-1.5228,0.0000
C00623=-67.616,-88.795,112.231,178.8242,-2.2388,0.0000
C00624=-61.928,-81.090,110.921,178.2745,-2.2660,0.0000
C00625=-55.342,-72.662,108.168,178.1738,-2.4056,0.0000
C00626=-49.111,-64.751,104.375,178.1836,-2.4208,0.0000
C00627=-44.239,-58.473,100.503,178.7380,-1.7453,0.0000
C00628=-41.961,-53.951,97.611,-179.2487,13.4881,0.0000
C00629=-43.616,-50.317,96.447,163.6122,21.2623,0.0000
C00630=-45.644,-48.318,96.396,159.5592,19.2137,0.0000
C00631=-46.992,-46.992,96.430,160.1702,19.8289,0.0000
C00632=-48.317,-45.644,96.396,160.7867,20.4413,0.0000
C00633=-50.318,-43.616,96.447,158.7369,16.3854,0.0000
C00634=-53.952,-41.961,97.611,166.5126,-0.7516,0.0000
C00635=-58.473,-44.239,100.503,-178.2547,1.2620,0.0000
C00636=-64.751,-49.111,104.375,-177.5792,1.8164,0.0000
C00637=-72.662,-55.342,108.168,-177.5944,1.8262,0.0000
C00638=-81.090,-61.928,110.921,-177.7340,1.7255,0.0000
C00639=-88.795,-67.616,112.231,-177.7612,1.1758,0.0000
C00640=-96.852,-69.288,112.908,-178.4772,-0.1213,0.0000
C00641=-104.285,-66.607,113.453,-179.4285,-0.4038,0.0000
C00642=-109.570,-60.156,113.997,-179.9789,-0.0383,0.0000
C00643=-113.636,-52.074,114.352,-179.9980,-0.0044,0.0000
C00644=-117.175,-43.531,114.352,-179.9983,-0.0046,0.0000
C00645=-120.015,-34.941,113.997,-179.9878,-0.0420,0.0000
C00646=-120.839,-26.642,113.453,179.8814,-0.6896,0.0000
C00647=-117.478,-19.491,112.908,179.0088,-1.1626,0.0000
C00648=-110.600,-14.976,112.231,177.5861,-0.7523,0.0000
C00649=-101.129,-13.549,110.921,177.1787,-0.3827,0.0000
C00650=-90.513,-12.247,108.168,177.0090,-0.4102,0.0000
C00651=-80.512,-11.059,104.375,177.0051,-0.4279,0.0000
C00652=-72.628,-10.065,100.503,177.8739,-0.3420,0.0000
C00653=-67.820,-8.479,97.611,-169.8583,9.1089,0.0000
C00654=-66.421,-4.738,96.447,-176.1552,25.7853,0.0000
C00655=-66.441,-1.891,96.396,179.0196,27.0204,0.0000
C00656=-66.457,0.000,96.430,179.9993,27.0201,0.0000
C00657=-66.441,1.890,96.396,-179.0188,27.0205,0.0000
C00658=-66.421,4.739,96.447,176.1528,25.7844,0.0000
C00659=-67.820,8.479,97.611,169.8585,9.1082,0.0000
C00660=-72.628,10.065,100.503,-177.8739,-0.3420,0.0000
C00661=-80.512,11.059,104.375,-177.0051,-0.4279,0.0000
C00662=-90.513,12.247,108.168,-177.0090,-0.4102,0.0000
C00663=-101.129,13.549,110.921,-177.1787,-0.3827,0.0000
C00664=-110.600,14.976,112.231,-177.5861,-0.7523,0.0000
C00665=-117.478,19.491,112.908,-179.0088,-1.1626,0.0000
C00666=-120.839,26.642,113.453,-179.8814,-0.6896,0.0000
C00667=-120.015,34.941,113.997,179.9878,-0.0420,0.0000
C00668=-117.175,43.531,114.352,179.9983,-0.0046,0.0000
C00669=-113.636,52.074,114.352,179.9980,-0.0044,0.0000
C00670=-109.570,60.156,113.997,179.9789,-0.0383,0.0000
C00671=-104.285,66.607,113.453,179.4285,-0.4038,0.0000
C00672=-96.852,69.288,112.908,178.4772,-0.1213,0.0000
C00673=-88.795,67.616,112.231,177.7612,1.1758,0.0000
C00674=-81.090,61.928,110.921,177.7340,1.7255,0.0000
C00675=-72.662,55.342,108.168,177.5944,1.8262,0.0000
C00676=-64.751,49.111,104.375,177.5792,1.8164,0.0000
C00677=-58.473,44.239,100.503,178.2547,1.2620,0.0000
C00678=-53.951,41.961,97.611,-166.5119,-0.7513,0.0000
C00679=-50.317,43.616,96.447,-158.7377,16.3878,0.0000
C00680=-48.318,45.644,96.396,-160.7863,20.4408,0.0000
C00681=-46.992,46.992,96.430,-160.1711,19.8298,0.0000
C00682=-45.644,48.317,96.396,-159.5587,19.2133,0.0000
C00683=-43.616,50.318,96.447,-163.6146,21.2631,0.0000
C00684=-41.961,53.952,97.611,179.2484,13.4874,0.0000
C00685=-44.239,58.473,100.503,-178.7380,-1.7453,0.0000
C00686=-49.111,64.751,104.375,-178.1836,-2.4208,0.0000
C00687=-55.342,72.662,108.168,-178.1738,-2.4056,0.0000
C00688=-61.928,81.090,110.921,-178.2745,-2.2660,0.0000
C00689=-67.616,88.795,112.231,-178.8242,-2.2388,0.0000
C00690=-69.288,96.852,112.908,179.8787,-1.5228,0.0000
C00691=-66.607,104.285,113.453,179.5962,-0.5715,0.0000
C00692=-60.156,109.570,113.997,179.9617,-0.0211,0.0000
C00693=-52.074,113.636,114.352,179.9956,-0.0020,0.0000
C00694=-43.531,117.175,114.352,179.9954,-0.0017,0.0000
C00695=-34.941,120.015,113.997,179.9580,-0.0122,0.0000
C00696=-26.642,120.839,113.453,179.3104,0.1186,0.0000
C00697=-19.491,117.478,112.908,178.8374,0.9912,0.0000
C00698=-14.976,110.600,112.231,179.2477,2.4139,0.0000
C00699=-13.549,101.129,110.921,179.6173,2.8213,0.0000
C00700=-12.247,90.513,108.168,179.5898,2.9910,0.0000
C00701=-11.059,80.512,104.375,179.5721,2.9949,0.0000
C00702=-10.065,72.628,100.503,179.6580,2.1261,0.0000
C00703=-8.479,67.820,97.611,-170.8918,-10.1415,0.0000
C00704=-4.739,66.421,96.447,-154.2156,-3.8472,0.0000
C00705=-1.890,66.441,96.396,-152.9795,0.9812,0.0000
C00706=0.000,66.457,96.430,-152.9799,-0.0007,0.0000
C00707=0.000,65.484,98.403,-154.5377,-0.0007,0.0000
C00708=1.802,65.470,98.368,-154.5345,-0.8753,0.0000
C00709=4.589,65.460,98.420,-155.7900,3.7631,0.0000
C00710=8.303,66.929,99.614,-171.8345,9.3277,0.0000
C00711=9.874,71.907,102.573,179.6823,-2.0507,0.0000
C00712=10.881,80.018,106.512,179.6257,-2.6726,0.0000
C00713=12.102,90.229,110.345,179.6614,-2.5019,0.0000
C00714=13.433,100.991,113.114,179.7069,-2.1881,0.0000
C00715=14.870,110.542,114.427,179.4526,-1.7704,0.0000
C00716=19.401,117.468,115.106,179.1811,-0.7010,0.0000
C00717=26.578,120.851,115.652,179.5319,-0.0810,0.0000
C00718=34.904,120.027,116.196,179.9728,0.0079,0.0000
C00719=43.519,117.179,116.552,179.9972,0.0011,0.0000
C00720=52.086,113.631,116.552,179.9972,0.0013,0.0000
C00721=60.191,109.553,116.196,179.9752,0.0136,0.0000
C00722=66.661,104.248,115.652,179.7263,0.3883,0.0000
C00723=69.344,96.781,115.106,179.9166,1.0747,0.0000
C00724=67.651,88.679,114.427,-179.1349,1.6389,0.0000
C00725=61.913,80.909,113.114,-178.6595,1.7547,0.0000
C00726=55.244,72.359,110.345,-178.4696,2.0088,0.0000
C00727=48.887,64.275,106.512,-178.3739,2.1548,0.0000
C00728=43.864,57.827,102.573,-178.7742,1.6749,0.0000
C00729=41.455,53.197,99.614,179.1587,-12.2765,0.0000
C00730=43.043,49.532,98.420,-164.8143,-20.0240,0.0000
C00731=45.020,47.568,98.368,-160.8349,-18.0533,0.0000
C00732=46.304,46.304,98.403,-161.3911,-18.6080,0.0000
C00733=47.568,45.021,98.368,-161.9471,-19.1655,0.0000
C00734=49.533,43.042,98.420,-159.9753,-15.1834,0.0000
C00735=53.197,41.455,99.614,-167.7243,0.8416,0.0000
C00736=57.827,43.864,102.573,178.3251,-1.2258,0.0000
C00737=64.275,48.887,106.512,177.8452,-1.6261,0.0000
C00738=72.359,55.244,110.345,177.9912,-1.5304,0.0000
C00739=80.909,61.913,113.114,178.2453,-1.3405,0.0000
C00740=88.679,67.651,114.427,178.3611,-0.8651,0.0000
C00741=96.781,69.344,115.106,178.9253,0.0834,0.0000
C00742=104.248,66.661,115.652,179.6117,0.2737,0.0000
C00743=109.553,60.191,116.196,179.9864,0.0248,0.0000
C00744=113.631,52.086,116.552,179.9987,0.0028,0.0000
C00745=117.179,43.519,116.552,179.9989,0.0028,0.0000
C00746=120.027,34.904,116.196,179.9921,0.0272,0.0000
C00747=120.851,26.578,115.652,-179.9190,0.4681,0.0000
C00748=117.468,19.401,115.106,-179.2990,0.8189,0.0000
C00749=110.542,14.870,114.427,-178.2296,0.5474,0.0000
C00750=100.991,13.433,113.114,-177.8119,0.2931,0.0000
C00751=90.229,12.102,110.345,-177.4981,0.3386,0.0000
C00752=80.018,10.881,106.512,-177.3274,0.3743,0.0000
C00753=71.907,9.874,102.573,-177.9493,0.3177,0.0000
C00754=66.929,8.303,99.614,170.6723,-8.1655,0.0000
C00755=65.460,4.589,98.420,176.2369,-24.2100,0.0000
C00756=65.470,1.802,98.368,-179.1247,-25.4655,0.0000
C00757=65.484,0.000,98.403,-179.9993,-25.4623,0.0000
C00758=65.470,-1.801,98.368,179.1241,-25.4656,0.0000
C00759=65.460,-4.589,98.420,-176.2346,-24.2091,0.0000
C00760=66.929,-8.303,99.614,-170.6726,-8.1647,0.0000
C00761=71.907,-9.874,102.573,177.9493,0.3177,0.0000
C00762=80.018,-10.881,106.512,177.3274,0.3743,0.0000
C00763=90.229,-12.102,110.345,177.4981,0.3386,0.0000
C00764=100.991,-13.433,113.114,177.8119,0.2931,0.0000
C00765=110.542,-14.870,114.427,178.2296,0.5474,0.0000
C00766=117.468,-19.401,115.106,179.2990,0.8189,0.0000
C00767=120.851,-26.578,115.652,179.9190,0.4681,0.0000
C00768=120.027,-34.904,116.196,-179.9921,0.0272,0.0000
C00769=117.179,-43.519,116.552,-179.9989,0.0028,0.0000
C00770=113.631,-52.086,116.552,-179.9987,0.0028,0.0000
C00771=109.553,-60.191,116.196,-179.9864,0.0248,0.0000
C00772=104.248,-66.661,115.652,-179.6117,0.2737,0.0000
C00773=96.781,-69.344,115.106,-178.9253,0.0834,0.0000
C00774=88.679,-67.651,114.427,-178.3611,-0.8651,0.0000
C00775=80.909,-61.913,113.114,-178.2453,-1.3405,0.0000
C00776=72.359,-55.244,110.345,-177.9912,-1.5304,0.0000
C00777=64.275,-48.887,106.512,-177.8452,-1.6261,0.0000
C00778=57.827,-43.864,102.573,-178.3251,-1.2258,0.0000
C00779=53.197,-41.455,99.614,167.7235,0.8413,0.0000
C00780=49.532,-43.043,98.420,159.9760,-15.1857,0.0000
C00781=47.568,-45.020,98.368,161.9467,-19.1651,0.0000
C00782=46.304,-46.304,98.403,161.3920,-18.6089,0.0000
C00783=45.021,-47.568,98.368,160.8345,-18.0529,0.0000
C00784=43.042,-49.533,98.420,164.8166,-20.0247,0.0000
C00785=41.455,-53.197,99.614,-179.1584,-12.2757,0.0000
C00786=43.864,-57.827,102.573,178.7742,1.6749,0.0000
C00787=48.887,-64.275,106.512,178.3739,2.1548,0.0000
C00788=55.244,-72.359,110.345,178.4696,2.0088,0.0000
C00789=61.913,-80.909,113.114,178.6595,1.7547,0.0000
C00790=67.651,-88.679,114.427,179.1349,1.6389,0.0000
C00791=69.344,-96.781,115.106,-179.9166,1.0747,0.0000
C00792=66.661,-104.248,115.652,-179.7263,0.3883,0.0000
C00793=60.191,-109.553,116.196,-179.9752,0.0136,0.0000
C00794=52.086,-113.631,116.552,-179.9972,0.0013,0.0000
C00795=43.519,-117.179,116.552,-179.9972,0.0011,0.0000
C00796=34.904,-120.027,116.196,-179.9728,0.0079,0.0000
C00797=26.578,-120.851,115.652,-179.5319,-0.0810,0.0000
C00798=19.401,-117.468,115.106,-179.1811,-0.7010,0.0000
C00799=14.870,-110.542,114.427,-179.4526,-1.7704,0.0000
C00800=13.433,-100.991,113.114,-179.7069,-2.1881,0.0000
C00801=12.102,-90.229,110.345,-179.6614,-2.5019,0.0000
C00802=10.881,-80.018,106.512,-179.6257,-2.6726,0.0000
C00803=9.874,-71.907,102.573,-179.6823,-2.0507,0.0000
C00804=8.303,-66.929,99.614,171.8345,9.3277,0.0000
C00805=4.589,-65.460,98.420,155.7900,3.7631,0.0000
C00806=1.802,-65.470,98.368,154.5345,-0.8753,0.0000
C00807=0.000,-65.484,98.403,154.5377,-0.0007,0.0000
C00808=0.000,-65.484,98.403,154.5377,-0.0007,0.0000
C00809=-1.801,-65.470,98.368,154.5344,0.8759,0.0000
C00810=-4.589,-65.460,98.420,155.7909,-3.7654,0.0000
C00811=-8.303,-66.929,99.614,171.8353,-9.3274,0.0000
C00812=-9.874,-71.907,102.573,-179.6823,2.0507,0.0000
C00813=-10.881,-80.018,106.512,-179.6257,2.6726,0.0000
C00814=-12.102,-90.229,110.345,-179.6614,2.5019,0.0000
C00815=-13.433,-100.991,113.114,-179.7069,2.1881,0.0000
C00816=-14.870,-110.542,114.427,-179.4526,1.7704,0.0000
C00817=-19.401,-117.468,115.106,-179.1811,0.7010,0.0000
C00818=-26.578,-120.851,115.652,-179.5319,0.0810,0.0000
C00819=-34.904,-120.027,116.196,-179.9728,-0.0079,0.0000
C00820=-43.519,-117.179,116.552,-179.9972,-0.0011,0.0000
C00821=-52.086,-113.631,116.552,-179.9972,-0.0013,0.0000
C00822=-60.191,-109.553,116.196,-179.9752,-0.0136,0.0000
C00823=-66.661,-104.248,115.652,-179.7263,-0.3883,0.0000
C00824=-69.344,-96.781,115.106,-179.9166,-1.0747,0.0000
C00825=-67.651,-88.679,114.427,179.1349,-1.6389,0.0000
C00826=-61.913,-80.909,113.114,178.6595,-1.7547,0.0000
C00827=-55.244,-72.359,110.345,178.4696,-2.0088,0.0000
C00828=-48.887,-64.275,106.512,178.3739,-2.1548,0.0000
C00829=-43.864,-57.827,102.573,178.7742,-1.6749,0.0000
C00830=-41.455,-53.197,99.614,-179.1587,12.2765,0.0000
C00831=-43.043,-49.532,98.420,164.8143,20.0240,0.0000
C00832=-45.020,-47.568,98.368,160.8349,18.0533,0.0000
C00833=-46.304,-46.304,98.403,161.3911,18.6080,0.0000
C00834=-47.568,-45.021,98.368,161.9471,19.1655,0.0000
C00835=-49.533,-43.042,98.420,159.9753,15.1834,0.0000
C00836=-53.197,-41.455,99.614,167.7243,-0.8416,0.0000
C00837=-57.827,-43.864,102.573,-178.3251,1.2258,0.0000
C00838=-64.275,-48.887,106.512,-177.8452,1.6261,0.0000
C00839=-72.359,-55.244,110.345,-177.9912,1.5304,0.0000
C00840=-80.909,-61.913,113.114,-178.2453,1.3405,0.0000
C00841=-88.679,-67.651,114.427,-178.3611,0.8651,0.0000
C00842=-96.781,-69.344,115.106,-178.9253,-0.0834,0.0000
C00843=-104.248,-66.661,115.652,-179.6117,-0.2737,0.0000
C00844=-109.553,-60.191,116.196,-179.9864,-0.0248,0.0000
C00845=-113.631,-52.086,116.552,-179.9987,-0.0028,0.0000
C00846=-117.179,-43.519,116.552,-179.9989,-0.0028,0.0000
C00847=-120.027,-34.904,116.196,-179.9921,-0.0272,0.0000
C00848=-120.851,-26.578,115.652,179.9190,-0.4681,0.0000
C00849=-117.468,-19.401,115.106,179.2990,-0.8189,0.0000
C00850=-110.542,-14.870,114.427,178.2296,-0.5474,0.0000
C00851=-100.991,-13.433,113.114,177.8119,-0.2931,0.0000
C00852=-90.229,-12.102,110.345,177.4981,-0.3386,0.0000
C00853=-80.018,-10.881,106.512,177.3274,-0.3743,0.0000
C00854=-71.907,-9.874,102.573,177.9493,-0.3177,0.0000
C00855=-66.929,-8.303,99.614,-170.6723,8.1655,0.0000
C00856=-65.460,-4.589,98.420,-176.2369,24.2100,0.0000
C00857=-65.470,-1.802,98.368,179.1247,25.4655,0.0000
C00858=-65.484,0.000,98.403,179.9993,25.4623,0.0000
C00859=-65.470,1.801,98.368,-179.1241,25.4656,0.0000
C00860=-65.460,4.589,98.420,176.2346,24.2091,0.0000
C00861=-66.929,8.303,99.614,170.6726,8.1647,0.0000
C00862=-71.907,9.874,102.573,-177.9493,-0.3177,0.0000
C00863=-80.018,10.881,106.512,-177.3274,-0.3743,0.0000
C00864=-90.229,12.102,110.345,-177.4981,-0.3386,0.0000
C00865=-100.991,13.433,113.114,-177.8119,-0.2931,0.0000
C00866=-110.542,14.870,114.427,-178.2296,-0.5474,0.0000
C00867=-117.468,19.401,115.106,-179.2990,-0.8189,0.0000
C00868=-120.851,26.578,115.652,-179.9190,-0.4681,0.0000
C00869=-120.027,34.904,116.196,179.9921,-0.0272,0.0000
C00870=-117.179,43.519,116.552,179.9989,-0.0028,0.0000
C00871=-113.631,52.086,116.552,179.9987,-0.0028,0.0000
C00872=-109.553,60.191,116.196,179.9864,-0.0248,0.0000
C00873=-104.248,66.661,115.652,179.6117,-0.2737,0.0000
C00874=-96.781,69.344,115.106,178.9253,-0.0834,0.0000
C00875=-88.679,67.651,114.427,178.3611,0.8651,0.0000
C00876=-80.909,61.913,113.114,178.2453,1.3405,0.0000
C00877=-72.359,55.244,110.345,177.9912,1.5304,0.0000
C00878=-64.275,48.887,106.512,177.8452,1.6261,0.0000
C00879=-57.827,43.864,102.573,178.3251,1.2258,0.0000
C00880=-53.197,41.455,99.614,-167.7235,-0.8413,0.0000
C00881=-49.532,43.043,98.420,-159.9760,15.1857,0.0000
C00882=-47.568,45.020,98.368,-161.9467,19.1651,0.0000
C00883=-46.304,46.304,98.403,-161.3920,18.6089,0.0000
C00884=-45.021,47.568,98.368,-160.8345,18.0529,0.0000
C00885=-43.042,49.533,98.420,-164.8166,20.0247,0.0000
C00886=-41.455,53.197,99.614,179.1584,12.2757,0.0000
C00887=-43.864,57.827,102.573,-178.7742,-1.6749,0.0000
C00888=-48.887,64.275,106.512,-178.3739,-2.1548,0.0000
C00889=-55.244,72.359,110.345,-178.4696,-2.0088,0.0000
C00890=-61.913,80.909,113.114,-178.6595,-1.7547,0.0000
C00891=-67.651,88.679,114.427,-179.1349,-1.6389,0.0000
C00892=-69.344,96.781,115.106,179.9166,-1.0747,0.0000
C00893=-66.661,104.248,115.652,179.7263,-0.3883,0.0000
C00894=-60.191,109.553,116.196,179.9752,-0.0136,0.0000
C00895=-52.086,113.631,116.552,179.9972,-0.0013,0.0000
C00896=-43.519,117.179,116.552,179.9972,-0.0011,0.0000
C00897=-34.904,120.027,116.196,179.9728,-0.0079,0.0000
C00898=-26.578,120.851,115.652,179.5319,0.0810,0.0000
C00899=-19.401,117.468,115.106,179.1811,0.7010,0.0000
C00900=-14.870,110.542,114.427,179.4526,1.7704,0.0000
C00901=-13.433,100.991,113.114,179.7069,2.1881,0.0000
C00902=-12.102,90.229,110.345,179.6614,2.5019,0.0000
C00903=-10.881,80.018,106.512,179.6257,2.6726,0.0000
C00904=-9.874,71.907,102.573,179.6823,2.0507,0.0000
C00905=-8.303,66.929,99.614,-171.8353,-9.3274,0.0000
C00906=-4.589,65.460,98.420,-155.7909,-3.7654,0.0000
C00907=-1.801,65.470,98.368,-154.5344,0.8759,0.0000
C00908=0.000,65.484,98.403,-154.5377,-0.0007,0.0000
C00909=0.000,64.567,100.403,-156.2412,-0.0006,0.0000
C00910=1.718,64.555,100.367,-156.2347,-0.7711,0.0000
C00911=4.448,64.555,100.420,-157.4947,3.6318,0.0000
C00912=8.138,66.095,101.644,-172.7502,8.4816,0.0000
C00913=9.699,71.247,104.664,179.7112,-1.9297,0.0000
C00914=10.725,79.585,108.663,179.6813,-2.3165,0.0000
C00915=11.984,89.998,112.530,179.7347,-1.9815,0.0000
C00916=13.346,100.888,115.310,179.7980,-1.5221,0.0000
C00917=14.797,110.503,116.626,179.6633,-1.0946,0.0000
C00918=19.343,117.461,117.305,179.5402,-0.3947,0.0000
C00919=26.538,120.858,117.851,179.7639,-0.0410,0.0000
C00920=34.883,120.034,118.396,179.9883,0.0034,0.0000
C00921=43.513,117.182,118.752,179.9989,0.0004,0.0000
C00922=52.091,113.628,118.752,179.9990,0.0005,0.0000
C00923=60.210,109.543,118.396,179.9893,0.0059,0.0000
C00924=66.694,104.225,117.851,179.8621,0.1959,0.0000
C00925=69.380,96.735,117.305,179.9539,0.6042,0.0000
C00926=67.674,88.600,116.626,-179.4640,1.0121,0.0000
C00927=61.901,80.776,115.310,-179.0664,1.2192,0.0000
C00928=55.165,72.112,112.530,-178.7861,1.5888,0.0000
C00929=48.691,63.859,108.663,-178.5868,1.8636,0.0000
C00930=43.521,57.238,104.664,-178.8393,1.5689,0.0000
C00931=40.982,52.491,101.644,179.1124,-11.0563,0.0000
C00932=42.502,48.793,100.420,-166.0669,-18.6676,0.0000
C00933=44.433,46.862,100.367,-162.2097,-16.7961,0.0000
C00934=45.656,45.656,100.403,-162.7101,-17.2891,0.0000
C00935=46.862,44.433,100.367,-163.2043,-17.7906,0.0000
C00936=48.793,42.502,100.421,-161.3318,-13.9309,0.0000
C00937=52.491,40.982,101.644,-168.9445,0.8879,0.0000
C00938=57.238,43.521,104.664,178.4311,-1.1607,0.0000
C00939=63.859,48.691,108.663,178.1364,-1.4132,0.0000
C00940=72.112,55.165,112.530,178.4112,-1.2139,0.0000
C00941=80.776,61.901,115.310,178.7808,-0.9336,0.0000
C00942=88.600,67.674,116.626,178.9879,-0.5360,0.0000
C00943=96.735,69.380,117.305,179.3958,0.0461,0.0000
C00944=104.225,66.694,117.851,179.8041,0.1379,0.0000
C00945=109.543,60.210,118.396,179.9941,0.0107,0.0000
C00946=113.628,52.091,118.752,179.9995,0.0010,0.0000
C00947=117.182,43.513,118.752,179.9996,0.0011,0.0000
C00948=120.034,34.883,118.396,179.9966,0.0117,0.0000
C00949=120.858,26.538,117.851,-179.9590,0.2361,0.0000
C00950=117.461,19.343,117.305,-179.6053,0.4598,0.0000
C00951=110.503,14.797,116.626,-178.9054,0.3367,0.0000
C00952=100.888,13.346,115.310,-178.4779,0.2020,0.0000
C00953=89.998,11.984,112.530,-178.0185,0.2653,0.0000
C00954=79.585,10.725,108.663,-177.6835,0.3187,0.0000
C00955=71.247,9.699,104.664,-178.0703,0.2888,0.0000
C00956=66.095,8.138,101.644,171.5184,-7.2498,0.0000
C00957=64.555,4.448,100.420,176.3682,-22.5053,0.0000
C00958=64.555,1.718,100.367,-179.2289,-23.7653,0.0000
C00959=64.567,0.000,100.403,-179.9994,-23.7588,0.0000
C00960=64.555,-1.717,100.367,179.2283,-23.7653,0.0000
C00961=64.556,-4.448,100.421,-176.3661,-22.5043,0.0000
C00962=66.096,-8.139,101.644,-171.5187,-7.2491,0.0000
C00963=71.247,-9.699,104.664,178.0703,0.2888,0.0000
C00964=79.585,-10.725,108.663,177.6835,0.3187,0.0000
C00965=89.998,-11.984,112.530,178.0185,0.2653,0.0000
C00966=100.888,-13.346,115.310,178.4779,0.2020,0.0000
C00967=110.503,-14.797,116.626,178.9054,0.3367,0.0000
C00968=117.461,-19.343,117.305,179.6053,0.4598,0.0000
C00969=120.858,-26.538,117.851,179.9590,0.2361,0.0000
C00970=120.034,-34.883,118.396,-179.9966,0.0117,0.0000
C00971=117.182,-43.513,118.752,-179.9996,0.0011,0.0000
C00972=113.628,-52.091,118.752,-179.9995,0.0010,0.0000
C00973=109.543,-60.210,118.396,-179.9941,0.0107,0.0000
C00974=104.225,-66.694,117.851,-179.8041,0.1379,0.0000
C00975=96.735,-69.380,117.305,-179.3958,0.0461,0.0000
C00976=88.600,-67.674,116.626,-178.9879,-0.5360,0.0000
C00977=80.776,-61.901,115.310,-178.7808,-0.9336,0.0000
C00978=72.112,-55.165,112.530,-178.4112,-1.2139,0.0000
C00979=63.859,-48.691,108.663,-178.1364,-1.4132,0.0000
C00980=57.238,-43.521,104.664,-178.4311,-1.1607,0.0000
C00981=52.491,-40.982,101.644,168.9437,0.8876,0.0000
C00982=48.793,-42.502,100.420,161.3324,-13.9331,0.0000
C00983=46.862,-44.433,100.367,163.2039,-17.7903,0.0000
C00984=45.656,-45.656,100.403,162.7109,-17.2899,0.0000
C00985=44.433,-46.862,100.367,162.2094,-16.7957,0.0000
C00986=42.502,-48.793,100.421,166.0691,-18.6682,0.0000
C00987=40.982,-52.491,101.644,-179.1121,-11.0555,0.0000
C00988=43.521,-57.238,104.664,178.8393,1.5689,0.0000
C00989=48.691,-63.859,108.663,178.5868,1.8636,0.0000
C00990=55.165,-72.112,112.530,178.7861,1.5888,0.0000
C00991=61.901,-80.776,115.310,179.0664,1.2192,0.0000
C00992=67.674,-88.600,116.626,179.4640,1.0121,0.0000
C00993=69.380,-96.735,117.305,-179.9539,0.6042,0.0000
C00994=66.694,-104.225,117.851,-179.8621,0.1959,0.0000
C00995=60.210,-109.543,118.396,-179.9893,0.0059,0.0000
C00996=52.091,-113.628,118.752,-179.9990,0.0005,0.0000
C00997=43.513,-117.182,118.752,-179.9989,0.0004,0.0000
C00998=34.883,-120.034,118.396,-179.9883,0.0034,0.0000
C00999=26.538,-120.858,117.851,-179.7639,-0.0410,0.0000
C01000=19.343,-117.461,117.305,-179.5402,-0.3947,0.0000
C01001=14.797,-110.503,116.626,-179.6633,-1.0946,0.0000
C01002=13.346,-100.888,115.310,-179.7980,-1.5221,0.0000
C01003=11.984,-89.998,112.530,-179.7347,-1.9815,0.0000
C01004=10.725,-79.585,108.663,-179.6813,-2.3165,0.0000
C01005=9.699,-71.247,104.664,-179.7112,-1.9297,0.0000
C01006=8.138,-66.095,101.644,172.7502,8.4816,0.0000
C01007=4.448,-64.555,100.420,157.4947,3.6318,0.0000
C01008=1.718,-64.555,100.367,156.2347,-0.7711,0.0000
C01009=0.000,-64.567,100.403,156.2412,-0.0006,0.0000
C01010=0.000,-64.567,100.403,156.2412,-0.0006,0.0000
C01011=-1.717,-64.555,100.367,156.2347,0.7717,0.0000
C01012=-4.448,-64.556,100.421,157.4957,-3.6339,0.0000
C01013=-8.139,-66.096,101.644,172.7509,-8.4813,0.0000
C01014=-9.699,-71.247,104.664,-179.7112,1.9297,0.0000
C01015=-10.725,-79.585,108.663,-179.6813,2.3165,0.0000
C01016=-11.984,-89.998,112.530,-179.7347,1.9815,0.0000
C01017=-13.346,-100.888,115.310,-179.7980,1.5221,0.0000
C01018=-14.797,-110.503,116.626,-179.6633,1.0946,0.0000
C01019=-19.343,-117.461,117.305,-179.5402,0.3947,0.0000
C01020=-26.538,-120.858,117.851,-179.7639,0.0410,0.0000
C01021=-34.883,-120.034,118.396,-179.9883,-0.0034,0.0000
C01022=-43.513,-117.182,118.752,-179.9989,-0.0004,0.0000
C01023=-52.091,-113.628,118.752,-179.9990,-0.0005,0.0000
C01024=-60.210,-109.543,118.396,-179.9893,-0.0059,0.0000
C01025=-66.694,-104.225,117.851,-179.8621,-0.1959,0.0000
C01026=-69.380,-96.735,117.305,-179.9539,-0.6042,0.0000
C01027=-67.674,-88.600,116.626,179.4640,-1.0121,0.0000
C01028=-61.901,-80.776,115.310,179.0664,-1.2192,0.0000
C01029=-55.165,-72.112,112.530,178.7861,-1.5888,0.0000
C01030=-48.691,-63.859,108.663,178.5868,-1.8636,0.0000
C01031=-43.521,-57.238,104.664,178.8393,-1.5689,0.0000
C01032=-40.982,-52.491,101.644,-179.1124,11.0563,0.0000
C01033=-42.502,-48.793,100.420,166.0669,18.6676,0.0000
C01034=-44.433,-46.862,100.367,162.2097,16.7961,0.0000
C01035=-45.656,-45.656,100.403,162.7101,17.2891,0.0000
C01036=-46.862,-44.433,100.367,163.2043,17.7906,0.0000
C01037=-48.793,-42.502,100.421,161.3318,13.9309,0.0000
C01038=-52.491,-40.982,101.644,168.9445,-0.8879,0.0000
C01039=-57.238,-43.521,104.664,-178.4311,1.1607,0.0000
C01040=-63.859,-48.691,108.663,-178.1364,1.4132,0.0000
C01041=-72.112,-55.165,112.530,-178.4112,1.2139,0.0000
C01042=-80.776,-61.901,115.310,-178.7808,0.9336,0.0000
C01043=-88.600,-67.674,116.626,-178.9879,0.5360,0.0000
C01044=-96.735,-69.380,117.305,-179.3958,-0.0461,0.0000
C01045=-104.225,-66.694,117.851,-179.8041,-0.1379,0.0000
C01046=-109.543,-60.210,118.396,-179.9941,-0.0107,0.0000
C01047=-113.628,-52.091,118.752,-179.9995,-0.0010,0.0000
C01048=-117.182,-43.513,118.752,-179.9996,-0.0011,0.0000
C01049=-120.034,-34.883,118.396,-179.9966,-0.0117,0.0000
C01050=-120.858,-26.538,117.851,179.9590,-0.2361,0.0000
C01051=-117.461,-19.343,117.305,179.6053,-0.4598,0.0000
C01052=-110.503,-14.797,116.626,178.9054,-0.3367,0.0000
C01053=-100.888,-13.346,115.310,178.4779,-0.2020,0.0000
C01054=-89.998,-11.984,112.530,178.0185,-0.2653,0.0000
C01055=-79.585,-10.725,108.663,177.6835,-0.3187,0.0000
C01056=-71.247,-9.699,104.664,178.0703,-0.2888,0.0000
C01057=-66.095,-8.138,101.644,-171.5184,7.2498,0.0000
C01058=-64.555,-4.448,100.420,-176.3682,22.5053,0.0000
C01059=-64.555,-1.718,100.367,179.2289,23.7653,0.0000
C01060=-64.567,0.000,100.403,179.9994,23.7588,0.0000
C01061=-64.555,1.717,100.367,-179.2283,23.7653,0.0000
C01062=-64.556,4.448,100.421,176.3661,22.5043,0.0000
C01063=-66.096,8.139,101.644,171.5187,7.2491,0.0000
C01064=-71.247,9.699,104.664,-178.0703,-0.2888,0.0000
C01065=-79.585,10.725,108.663,-177.6835,-0.3187,0.0000
C01066=-89.998,11.984,112.530,-178.0185,-0.2653,0.0000
C01067=-100.888,13.346,115.310,-178.4779,-0.2020,0.0000
C01068=-110.503,14.797,116.626,-178.9054,-0.3367,0.0000
C01069=-117.461,19.343,117.305,-179.6053,-0.4598,0.0000
C01070=-120.858,26.538,117.851,-179.9590,-0.2361,0.0000
C01071=-120.034,34.883,118.396,179.9966,-0.0117,0.0000
C01072=-117.182,43.513,118.752,179.9996,-0.0011,0.0000
C01073=-113.628,52.091,118.752,179.9995,-0.0010,0.0000
C01074=-109.543,60.210,118.396,179.9941,-0.0107,0.0000
C01075=-104.225,66.694,117.851,179.8041,-0.1379,0.0000
C01076=-96.735,69.380,117.305,179.3958,-0.0461,0.0000
C01077=-88.600,67.674,116.626,178.9879,0.5360,0.0000
C01078=-80.776,61.901,115.310,178.7808,0.9336,0.0000
C01079=-72.112,55.165,112.530,178.4112,1.2139,0.0000
C01080=-63.859,48.691,108.663,178.1364,1.4132,0.0000
C01081=-57.238,43.521,104.664,178.4311,1.1607,0.0000
C01082=-52.491,40.982,101.644,-168.9437,-0.8876,0.0000
C01083=-48.793,42.502,100.420,-161.3324,13.9331,0.0000
C01084=-46.862,44.433,100.367,-163.2039,17.7903,0.0000
C01085=-45.656,45.656,100.403,-162.7109,17.2899,0.0000
C01086=-44.433,46.862,100.367,-162.2094,16.7957,0.0000
C01087=-42.502,48.793,100.421,-166.0691,18.6682,0.0000
C01088=-40.982,52.491,101.644,179.1121,11.0555,0.0000
C01089=-43.521,57.238,104.664,-178.8393,-1.5689,0.0000
C01090=-48.691,63.859,108.663,-178.5868,-1.8636,0.0000
C01091=-55.165,72.112,112.530,-178.7861,-1.5888,0.0000
C01092=-61.901,80.776,115.310,-179.0664,-1.2192,0.0000
C01093=-67.674,88.600,116.626,-179.4640,-1.0121,0.0000
C01094=-69.380,96.735,117.305,179.9539,-0.6042,0.0000
C01095=-66.694,104.225,117.851,179.8621,-0.1959,0.0000
C01096=-60.210,109.543,118.396,179.9893,-0.0059,0.0000
C01097=-52.091,113.628,118.752,179.9990,-0.0005,0.0000
C01098=-43.513,117.182,118.752,179.9989,-0.0004,0.0000
C01099=-34.883,120.034,118.396,179.9883,-0.0034,0.0000
C01100=-26.538,120.858,117.851,179.7639,0.0410,0.0000
C01101=-19.343,117.461,117.305,179.5402,0.3947,0.0000
C01102=-14.797,110.503,116.626,179.6633,1.0946,0.0000
C01103=-13.346,100.888,115.310,179.7980,1.5221,0.0000
C01104=-11.984,89.998,112.530,179.7347,1.9815,0.0000
C01105=-10.725,79.585,108.663,179.6813,2.3165,0.0000
C01106=-9.699,71.247,104.664,179.7112,1.9297,0.0000
C01107=-8.139,66.096,101.644,-172.7509,-8.4813,0.0000
C01108=-4.448,64.556,100.421,-157.4957,-3.6339,0.0000
C01109=-1.717,64.555,100.367,-156.2347,0.7717,0.0000
C01110=0.000,64.567,100.403,-156.2412,-0.0006,0.0000
C01111=0.000,63.713,102.430,-158.1009,-0.0005,0.0000
C01112=1.640,63.703,102.394,-158.0906,-0.6691,0.0000
C01113=4.317,63.713,102.448,-159.3359,3.4482,0.0000
C01114=7.987,65.326,103.699,-173.6400,7.6051,0.0000
C01115=9.542,70.656,106.778,179.7440,-1.7650,0.0000
C01116=10.593,79.218,110.828,179.7386,-1.9280,0.0000
C01117=11.894,89.822,114.721,179.8100,-1.4313,0.0000
C01118=13.292,100.823,117.508,179.8911,-0.8249,0.0000
C01119=14.760,110.482,118.825,179.8808,-0.3886,0.0000
C01120=19.318,117.458,119.505,179.9140,-0.0739,0.0000
C01121=69.395,96.715,119.505,179.9914,0.1131,0.0000
C01122=67.686,88.559,118.825,-179.8095,0.3590,0.0000
C01123=61.894,80.692,117.508,-179.4936,0.6603,0.0000
C01124=55.104,71.924,114.721,-179.1222,1.1465,0.0000
C01125=48.525,63.506,110.828,-178.8212,1.5483,0.0000
C01126=43.214,56.709,106.778,-178.9327,1.4292,0.0000
C01127=40.545,51.840,103.699,179.1064,-9.8277,0.0000
C01128=41.999,48.104,102.448,-167.3698,-17.1865,0.0000
C01129=43.885,46.204,102.394,-163.6880,-15.4365,0.0000
C01130=45.052,45.052,102.430,-164.1323,-15.8671,0.0000
C01131=46.204,43.886,102.394,-164.5638,-16.3122,0.0000
C01132=48.104,41.999,102.448,-162.8129,-12.6281,0.0000
C01133=51.840,40.545,103.699,-170.1730,0.8939,0.0000
C01134=56.709,43.214,106.778,178.5708,-1.0673,0.0000
C01135=63.506,48.525,110.828,178.4517,-1.1788,0.0000
C01136=71.924,55.104,114.721,178.8535,-0.8778,0.0000
C01137=80.692,61.894,117.508,179.3397,-0.5064,0.0000
C01138=88.559,67.686,118.825,179.6410,-0.1905,0.0000
C01139=96.715,69.395,119.505,179.8869,0.0086,0.0000
C01140=117.458,19.318,119.505,-179.9261,0.0860,0.0000
C01141=110.482,14.760,118.825,-179.6114,0.1192,0.0000
C01142=100.823,13.292,117.508,-179.1751,0.1089,0.0000
C01143=89.822,11.894,114.721,-178.5687,0.1900,0.0000
C01144=79.218,10.593,110.828,-178.0720,0.2614,0.0000
C01145=70.656,9.542,106.778,-178.2350,0.2560,0.0000
C01146=65.326,7.987,103.699,172.3949,-6.3600,0.0000
C01147=63.713,4.317,102.448,176.5518,-20.6641,0.0000
C01148=63.703,1.640,102.394,-179.3309,-21.9094,0.0000
C01149=63.713,0.000,102.430,-179.9995,-21.8991,0.0000
C01150=63.703,-1.639,102.394,179.3305,-21.9094,0.0000
C01151=63.713,-4.317,102.448,-176.5498,-20.6631,0.0000
C01152=65.326,-7.987,103.699,-172.3952,-6.3593,0.0000
C01153=70.656,-9.542,106.778,178.2350,0.2560,0.0000
C01154=79.218,-10.593,110.828,178.0720,0.2614,0.0000
C01155=89.822,-11.894,114.721,178.5687,0.1900,0.0000
C01156=100.823,-13.292,117.508,179.1751,0.1089,0.0000
C01157=110.482,-14.760,118.825,179.6114,0.1192,0.0000
C01158=117.458,-19.318,119.505,179.9261,0.0860,0.0000
C01159=96.715,-69.395,119.505,-179.8869,0.0086,0.0000
C01160=88.559,-67.686,118.825,-179.6410,-0.1905,0.0000
C01161=80.692,-61.894,117.508,-179.3397,-0.5064,0.0000
C01162=71.924,-55.104,114.721,-178.8535,-0.8778,0.0000
C01163=63.506,-48.525,110.828,-178.4517,-1.1788,0.0000
C01164=56.709,-43.214,106.778,-178.5708,-1.0673,0.0000
C01165=51.840,-40.545,103.699,170.1723,0.8936,0.0000
C01166=48.104,-41.999,102.448,162.8135,-12.6302,0.0000
C01167=46.204,-43.885,102.394,164.5635,-16.3120,0.0000
C01168=45.052,-45.052,102.430,164.1329,-15.8677,0.0000
C01169=43.886,-46.204,102.394,163.6878,-15.4362,0.0000
C01170=41.999,-48.104,102.448,167.3719,-17.1871,0.0000
C01171=40.545,-51.840,103.699,-179.1061,-9.8270,0.0000
C01172=43.214,-56.709,106.778,178.9327,1.4292,0.0000
C01173=48.525,-63.506,110.828,178.8212,1.5483,0.0000
C01174=55.104,-71.924,114.721,179.1222,1.1465,0.0000
C01175=61.894,-80.692,117.508,179.4936,0.6603,0.0000
C01176=67.686,-88.559,118.825,179.8095,0.3590,0.0000
C01177=69.395,-96.715,119.505,-179.9914,0.1131,0.0000
C01178=19.318,-117.458,119.505,-179.9140,-0.0739,0.0000
C01179=14.760,-110.482,118.825,-179.8808,-0.3886,0.0000
C01180=13.292,-100.823,117.508,-179.8911,-0.8249,0.0000
C01181=11.894,-89.822,114.721,-179.8100,-1.4313,0.0000
C01182=10.593,-79.218,110.828,-179.7386,-1.9280,0.0000
C01183=9.542,-70.656,106.778,-179.7440,-1.7650,0.0000
C01184=7.987,-65.326,103.699,173.6400,7.6051,0.0000
C01185=4.317,-63.713,102.448,159.3359,3.4482,0.0000
C01186=1.640,-63.703,102.394,158.0906,-0.6691,0.0000
C01187=0.000,-63.713,102.430,158.1009,-0.0005,0.0000
C01188=0.000,-63.713,102.430,158.1009,-0.0005,0.0000
C01189=-1.639,-63.703,102.394,158.0906,0.6695,0.0000
C01190=-4.317,-63.713,102.448,159.3369,-3.4502,0.0000
C01191=-7.987,-65.326,103.699,173.6407,-7.6048,0.0000
C01192=-9.542,-70.656,106.778,-179.7440,1.7650,0.0000
C01193=-10.593,-79.218,110.828,-179.7386,1.9280,0.0000
C01194=-11.894,-89.822,114.721,-179.8100,1.4313,0.0000
C01195=-13.292,-100.823,117.508,-179.8911,0.8249,0.0000
C01196=-14.760,-110.482,118.825,-179.8808,0.3886,0.0000
C01197=-19.318,-117.458,119.505,-179.9140,0.0739,0.0000
C01198=-69.395,-96.715,119.505,-179.9914,-0.1131,0.0000
C01199=-67.686,-88.559,118.825,179.8095,-0.3590,0.0000
C01200=-61.894,-80.692,117.508,179.4936,-0.6603,0.0000
C01201=-55.104,-71.924,114.721,179.1222,-1.1465,0.0000
C01202=-48.525,-63.506,110.828,178.8212,-1.5483,0.0000
C01203=-43.214,-56.709,106.778,178.9327,-1.4292,0.0000
C01204=-40.545,-51.840,103.699,-179.1064,9.8277,0.0000
C01205=-41.999,-48.104,102.448,167.3698,17.1865,0.0000
C01206=-43.885,-46.204,102.394,163.6880,15.4365,0.0000
C01207=-45.052,-45.052,102.430,164.1323,15.8671,0.0000
C01208=-46.204,-43.886,102.394,164.5638,16.3122,0.0000
C01209=-48.104,-41.999,102.448,162.8129,12.6281,0.0000
C01210=-51.840,-40.545,103.699,170.1730,-0.8939,0.0000
C01211=-56.709,-43.214,106.778,-178.5708,1.0673,0.0000
C01212=-63.506,-48.525,110.828,-178.4517,1.1788,0.0000
C01213=-71.924,-55.104,114.721,-178.8535,0.8778,0.0000
C01214=-80.692,-61.894,117.508,-179.3397,0.5064,0.0000
C01215=-88.559,-67.686,118.825,-179.6410,0.1905,0.0000
C01216=-96.715,-69.395,119.505,-179.8869,-0.0086,0.0000
C01217=-117.458,-19.318,119.505,179.9261,-0.0860,0.0000
C01218=-110.482,-14.760,118.825,179.6114,-0.1192,0.0000
C01219=-100.823,-13.292,117.508,179.1751,-0.1089,0.0000
C01220=-89.822,-11.894,114.721,178.5687,-0.1900,0.0000
C01221=-79.218,-10.593,110.828,178.0720,-0.2614,0.0000
C01222=-70.656,-9.542,106.778,178.2350,-0.2560,0.0000
C01223=-65.326,-7.987,103.699,-172.3949,6.3600,0.0000
C01224=-63.713,-4.317,102.448,-176.5518,20.6641,0.0000
C01225=-63.703,-1.640,102.394,179.3309,21.9094,0.0000
C01226=-63.713,0.000,102.430,179.9995,21.8991,0.0000
C01227=-63.703,1.639,102.394,-179.3305,21.9094,0.0000
C01228=-63.713,4.317,102.448,176.5498,20.6631,0.0000
C01229=-65.326,7.987,103.699,172.3952,6.3593,0.0000
C01230=-70.656,9.542,106.778,-178.2350,-0.2560,0.0000
C01231=-79.218,10.593,110.828,-178.0720,-0.2614,0.0000
C01232=-89.822,11.894,114.721,-178.5687,-0.1900,0.0000
C01233=-100.823,13.292,117.508,-179.1751,-0.1089,0.0000
C01234=-110.482,14.760,118.825,-179.6114,-0.1192,0.0000
C01235=-117.458,19.318,119.505,-179.9261,-0.0860,0.0000
C01236=-96.715,69.395,119.505,179.8869,-0.0086,0.0000
C01237=-88.559,67.686,118.825,179.6410,0.1905,0.0000
C01238=-80.692,61.894,117.508,179.3397,0.5064,0.0000
C01239=-71.924,55.104,114.721,178.8535,0.8778,0.0000
C01240=-63.506,48.525,110.828,178.4517,1.1788,0.0000
C01241=-56.709,43.214,106.778,178.5708,1.0673,0.0000
C01242=-51.840,40.545,103.699,-170.1723,-0.8936,0.0000
C01243=-48.104,41.999,102.448,-162.8135,12.6302,0.0000
C01244=-46.204,43.885,102.394,-164.5635,16.3120,0.0000
C01245=-45.052,45.052,102.430,-164.1329,15.8677,0.0000
C01246=-43.886,46.204,102.394,-163.6878,15.4362,0.0000
C01247=-41.999,48.104,102.448,-167.3719,17.1871,0.0000
C01248=-40.545,51.840,103.699,179.1061,9.8270,0.0000
C01249=-43.214,56.709,106.778,-178.9327,-1.4292,0.0000
C01250=-48.525,63.506,110.828,-178.8212,-1.5483,0.0000
C01251=-55.104,71.924,114.721,-179.1222,-1.1465,0.0000
C01252=-61.894,80.692,117.508,-179.4936,-0.6603,0.0000
C01253=-67.686,88.559,118.825,-179.8095,-0.3590,0.0000
C01254=-69.395,96.715,119.505,179.9914,-0.1131,0.0000
C01255=-19.318,117.458,119.505,179.9140,0.0739,0.0000
C01256=-14.760,110.482,118.825,179.8808,0.3886,0.0000
C01257=-13.292,100.823,117.508,179.8911,0.8249,0.0000
C01258=-11.894,89.822,114.721,179.8100,1.4313,0.0000
C01259=-10.593,79.218,110.828,179.7386,1.9280,0.0000
C01260=-9.542,70.656,106.778,179.7440,1.7650,0.0000
C01261=-7.987,65.326,103.699,-173.6407,-7.6048,0.0000
C01262=-4.317,63.713,102.448,-159.3369,-3.4502,0.0000
C01263=-1.639,63.703,102.394,-158.0906,0.6695,0.0000
C01264=0.000,63.713,102.430,-158.1009,-0.0005,0.0000
C01265=0.000,62.929,104.486,-160.1268,-0.0004,0.0000
C01266=1.568,62.919,104.448,-160.1124,-0.5703,0.0000
C01267=4.196,62.938,104.504,-161.3200,3.2108,0.0000
C01268=7.849,64.627,105.781,-174.5070,6.6994,0.0000
C01269=9.405,70.138,108.911,179.7800,-1.5589,0.0000
C01270=10.487,78.922,113.006,179.7979,-1.5091,0.0000
C01271=11.833,89.705,116.917,179.8874,-0.8532,0.0000
C01272=13.270,100.797,119.708,179.9870,-0.0985,0.0000
C01273=61.891,80.658,119.708,-179.9395,0.0788,0.0000
C01274=55.063,71.798,116.917,-179.4764,0.6829,0.0000
C01275=48.391,63.222,113.006,-179.0757,1.2101,0.0000
C01276=42.945,56.245,108.911,-179.0531,1.2579,0.0000
C01277=40.148,51.249,105.781,179.1373,-8.5900,0.0000
C01278=41.537,47.471,104.504,-168.7231,-15.5750,0.0000
C01279=43.382,45.599,104.448,-165.2737,-13.9692,0.0000
C01280=44.497,44.497,104.486,-165.6622,-14.3373,0.0000
C01281=45.599,43.382,104.448,-166.0310,-14.7265,0.0000
C01282=47.472,41.536,104.504,-164.4245,-11.2750,0.0000
C01283=51.249,40.149,105.781,-171.4107,0.8630,0.0000
C01284=56.245,42.945,108.911,178.7421,-0.9469,0.0000
C01285=63.222,48.391,113.006,178.7899,-0.9243,0.0000
C01286=71.798,55.063,116.917,179.3171,-0.5236,0.0000
C01287=80.658,61.891,119.708,179.9212,-0.0605,0.0000
C01288=100.797,13.270,119.708,-179.9015,0.0130,0.0000
C01289=89.705,11.833,116.917,-179.1468,0.1126,0.0000
C01290=78.922,10.487,113.006,-178.4909,0.2021,0.0000
C01291=70.138,9.405,108.911,-178.4411,0.2200,0.0000
C01292=64.627,7.849,105.781,173.3006,-5.4930,0.0000
C01293=62.938,4.196,104.504,176.7892,-18.6800,0.0000
C01294=62.919,1.568,104.448,-179.4297,-19.8876,0.0000
C01295=62.929,0.000,104.486,-179.9996,-19.8732,0.0000
C01296=62.919,-1.567,104.448,179.4294,-19.8876,0.0000
C01297=62.938,-4.197,104.504,-176.7874,-18.6791,0.0000
C01298=64.628,-7.849,105.781,-173.3009,-5.4923,0.0000
C01299=70.138,-9.405,108.911,178.4411,0.2200,0.0000
C01300=78.922,-10.487,113.006,178.4909,0.2021,0.0000
C01301=89.705,-11.833,116.917,179.1468,0.1126,0.0000
C01302=100.797,-13.270,119.708,179.9015,0.0130,0.0000
C01303=80.658,-61.891,119.708,-179.9212,-0.0605,0.0000
C01304=71.798,-55.063,116.917,-179.3171,-0.5236,0.0000
C01305=63.222,-48.391,113.006,-178.7899,-0.9243,0.0000
C01306=56.245,-42.945,108.911,-178.7421,-0.9469,0.0000
C01307=51.249,-40.148,105.781,171.4100,0.8627,0.0000
C01308=47.471,-41.537,104.504,164.4250,-11.2769,0.0000
C01309=45.599,-43.382,104.448,166.0308,-14.7263,0.0000
C01310=44.497,-44.497,104.486,165.6627,-14.3378,0.0000
C01311=43.382,-45.599,104.448,165.2735,-13.9690,0.0000
C01312=41.536,-47.472,104.504,168.7250,-15.5755,0.0000
C01313=40.149,-51.249,105.781,-179.1370,-8.5893,0.0000
C01314=42.945,-56.245,108.911,179.0531,1.2579,0.0000
C01315=48.391,-63.222,113.006,179.0757,1.2101,0.0000
C01316=55.063,-71.798,116.917,179.4764,0.6829,0.0000
C01317=61.891,-80.658,119.708,179.9395,0.0788,0.0000
C01318=13.270,-100.797,119.708,-179.9870,-0.0985,0.0000
C01319=11.833,-89.705,116.917,-179.8874,-0.8532,0.0000
C01320=10.487,-78.922,113.006,-179.7979,-1.5091,0.0000
C01321=9.405,-70.138,108.911,-179.7800,-1.5589,0.0000
C01322=7.849,-64.627,105.781,174.5070,6.6994,0.0000
C01323=4.196,-62.938,104.504,161.3200,3.2108,0.0000
C01324=1.568,-62.919,104.448,160.1124,-0.5703,0.0000
C01325=0.000,-62.929,104.486,160.1268,-0.0004,0.0000
C01326=0.000,-62.929,104.486,160.1268,-0.0004,0.0000
C01327=-1.567,-62.919,104.448,160.1124,0.5706,0.0000
C01328=-4.197,-62.938,104.504,161.3209,-3.2126,0.0000
C01329=-7.849,-64.628,105.781,174.5077,-6.6991,0.0000
C01330=-9.405,-70.138,108.911,-179.7800,1.5589,0.0000
C01331=-10.487,-78.922,113.006,-179.7979,1.5091,0.0000
C01332=-11.833,-89.705,116.917,-179.8874,0.8532,0.0000
C01333=-13.270,-100.797,119.708,-179.9870,0.0985,0.0000
C01334=-61.891,-80.658,119.708,179.9395,-0.0788,0.0000
C01335=-55.063,-71.798,116.917,179.4764,-0.6829,0.0000
C01336=-48.391,-63.222,113.006,179.0757,-1.2101,0.0000
C01337=-42.945,-56.245,108.911,179.0531,-1.2579,0.0000
C01338=-40.148,-51.249,105.781,-179.1373,8.5900,0.0000
C01339=-41.537,-47.471,104.504,168.7231,15.5750,0.0000
C01340=-43.382,-45.599,104.448,165.2737,13.9692,0.0000
C01341=-44.497,-44.497,104.486,165.6622,14.3373,0.0000
C01342=-45.599,-43.382,104.448,166.0310,14.7265,0.0000
C01343=-47.472,-41.536,104.504,164.4245,11.2750,0.0000
C01344=-51.249,-40.149,105.781,171.4107,-0.8630,0.0000
C01345=-56.245,-42.945,108.911,-178.7421,0.9469,0.0000
C01346=-63.222,-48.391,113.006,-178.7899,0.9243,0.0000
C01347=-71.798,-55.063,116.917,-179.3171,0.5236,0.0000
C01348=-80.658,-61.891,119.708,-179.9212,0.0605,0.0000
C01349=-100.797,-13.270,119.708,179.9015,-0.0130,0.0000
C01350=-89.705,-11.833,116.917,179.1468,-0.1126,0.0000
C01351=-78.922,-10.487,113.006,178.4909,-0.2021,0.0000
C01352=-70.138,-9.405,108.911,178.4411,-0.2200,0.0000
C01353=-64.627,-7.849,105.781,-173.3006,5.4930,0.0000
C01354=-62.938,-4.196,104.504,-176.7892,18.6800,0.0000
C01355=-62.919,-1.568,104.448,179.4297,19.8876,0.0000
C01356=-62.929,0.000,104.486,179.9996,19.8732,0.0000
C01357=-62.919,1.567,104.448,-179.4294,19.8876,0.0000
C01358=-62.938,4.197,104.504,176.7874,18.6791,0.0000
C01359=-64.628,7.849,105.781,173.3009,5.4923,0.0000
C01360=-70.138,9.405,108.911,-178.4411,-0.2200,0.0000
C01361=-78.922,10.487,113.006,-178.4909,-0.2021,0.0000
C01362=-89.705,11.833,116.917,-179.1468,-0.1126,0.0000
C01363=-100.797,13.270,119.708,-179.9015,-0.0130,0.0000
C01364=-80.658,61.891,119.708,179.9212,0.0605,0.0000
C01365=-71.798,55.063,116.917,179.3171,0.5236,0.0000
C01366=-63.222,48.391,113.006,178.7899,0.9243,0.0000
C01367=-56.245,42.945,108.911,178.7421,0.9469,0.0000
C01368=-51.249,40.148,105.781,-171.4100,-0.8627,0.0000
C01369=-47.471,41.537,104.504,-164.4250,11.2769,0.0000
C01370=-45.599,43.382,104.448,-166.0308,14.7263,0.0000
C01371=-44.497,44.497,104.486,-165.6627,14.3378,0.0000
C01372=-43.382,45.599,104.448,-165.2735,13.9690,0.0000
C01373=-41.536,47.472,104.504,-168.7250,15.5755,0.0000
C01374=-40.149,51.249,105.781,179.1370,8.5893,0.0000
C01375=-42.945,56.245,108.911,-179.0531,-1.2579,0.0000
C01376=-48.391,63.222,113.006,-179.0757,-1.2101,0.0000
C01377=-55.063,71.798,116.917,-179.4764,-0.6829,0.0000
C01378=-61.891,80.658,119.708,-179.9395,-0.0788,0.0000
C01379=-13.270,100.797,119.708,179.9870,0.0985,0.0000
C01380=-11.833,89.705,116.917,179.8874,0.8532,0.0000
C01381=-10.487,78.922,113.006,179.7979,1.5091,0.0000
C01382=-9.405,70.138,108.911,179.7800,1.5589,0.0000
C01383=-7.849,64.628,105.781,-174.5077,-6.6991,0.0000
C01384=-4.197,62.938,104.504,-161.3209,-3.2126,0.0000
C01385=-1.567,62.919,104.448,-160.1124,0.5706,0.0000
C01386=0.000,62.929,104.486,-160.1268,-0.0004,0.0000
C01387=0.000,62.220,106.568,-162.3278,-0.0003,0.0000
C01388=1.503,62.212,106.531,-162.3086,-0.4759,0.0000
C01389=4.087,62.239,106.587,-163.4522,2.9184,0.0000
C01390=7.726,64.006,107.888,-175.3550,5.7650,0.0000
C01391=9.288,69.700,111.064,179.8189,-1.3141,0.0000
C01392=10.407,78.701,115.193,179.8590,-1.0619,0.0000
C01393=11.804,89.648,119.116,179.9672,-0.2493,0.0000
C01394=55.044,71.737,119.116,-179.8469,0.1995,0.0000
C01395=48.291,63.009,115.193,-179.3487,0.8506,0.0000
C01396=42.718,55.853,111.064,-179.1987,1.0573,0.0000
C01397=39.796,50.723,107.888,179.2015,-7.3415,0.0000
C01398=41.119,46.900,106.587,-170.1267,-13.8281,0.0000
C01399=42.927,45.053,106.531,-166.9699,-12.3897,0.0000
C01400=43.996,43.996,106.568,-167.3037,-12.6959,0.0000
C01401=45.053,42.928,106.530,-167.6104,-13.0302,0.0000
C01402=46.900,41.119,106.587,-166.1714,-9.8715,0.0000
C01403=50.723,39.796,107.888,-172.6591,0.7987,0.0000
C01404=55.853,42.718,111.064,178.9427,-0.8013,0.0000
C01405=63.009,48.291,115.193,179.1494,-0.6513,0.0000
C01406=71.737,55.044,119.116,179.8005,-0.1531,0.0000
C01407=89.648,11.804,119.116,-179.7507,0.0328,0.0000
C01408=78.701,10.407,115.193,-178.9381,0.1410,0.0000
C01409=69.700,9.288,111.064,-178.6859,0.1811,0.0000
C01410=64.006,7.726,107.888,174.2350,-4.6450,0.0000
C01411=62.239,4.087,106.587,177.0816,-16.5478,0.0000
C01412=62.212,1.503,106.531,-179.5241,-17.6914,0.0000
C01413=62.220,0.000,106.568,-179.9997,-17.6722,0.0000
C01414=62.212,-1.502,106.530,179.5239,-17.6913,0.0000
C01415=62.239,-4.088,106.587,-177.0800,-16.5469,0.0000
C01416=64.006,-7.727,107.888,-174.2353,-4.6444,0.0000
C01417=69.700,-9.288,111.064,178.6859,0.1811,0.0000
C01418=78.701,-10.407,115.193,178.9381,0.1410,0.0000
C01419=89.648,-11.804,119.116,179.7507,0.0328,0.0000
C01420=71.737,-55.044,119.116,-179.8005,-0.1531,0.0000
C01421=63.009,-48.291,115.193,-179.1494,-0.6513,0.0000
C01422=55.853,-42.718,111.064,-178.9427,-0.8013,0.0000
C01423=50.723,-39.796,107.888,172.6585,0.7985,0.0000
C01424=46.900,-41.119,106.587,166.1719,-9.8733,0.0000
C01425=45.053,-42.927,106.531,167.6103,-13.0301,0.0000
C01426=43.996,-43.996,106.568,167.3041,-12.6963,0.0000
C01427=42.928,-45.053,106.530,166.9698,-12.3896,0.0000
C01428=41.119,-46.900,106.587,170.1285,-13.8286,0.0000
C01429=39.796,-50.723,107.888,-179.2013,-7.3409,0.0000
C01430=42.718,-55.853,111.064,179.1987,1.0573,0.0000
C01431=48.291,-63.009,115.193,179.3487,0.8506,0.0000
C01432=55.044,-71.737,119.116,179.8469,0.1995,0.0000
C01433=11.804,-89.648,119.116,-179.9672,-0.2493,0.0000
C01434=10.407,-78.701,115.193,-179.8590,-1.0619,0.0000
C01435=9.288,-69.700,111.064,-179.8189,-1.3141,0.0000
C01436=7.726,-64.006,107.888,175.3550,5.7650,0.0000
C01437=4.087,-62.239,106.587,163.4522,2.9184,0.0000
C01438=1.503,-62.212,106.531,162.3086,-0.4759,0.0000
C01439=0.000,-62.220,106.568,162.3278,-0.0003,0.0000
C01440=0.000,-62.220,106.568,162.3278,-0.0003,0.0000
C01441=-1.502,-62.212,106.530,162.3087,0.4761,0.0000
C01442=-4.088,-62.239,106.587,163.4531,-2.9200,0.0000
C01443=-7.727,-64.006,107.888,175.3556,-5.7647,0.0000
C01444=-9.288,-69.700,111.064,-179.8189,1.3141,0.0000
C01445=-10.407,-78.701,115.193,-179.8590,1.0619,0.0000
C01446=-11.804,-89.648,119.116,-179.9672,0.2493,0.0000
C01447=-55.044,-71.737,119.116,179.8469,-0.1995,0.0000
C01448=-48.291,-63.009,115.193,179.3487,-0.8506,0.0000
C01449=-42.718,-55.853,111.064,179.1987,-1.0573,0.0000
C01450=-39.796,-50.723,107.888,-179.2015,7.3415,0.0000
C01451=-41.119,-46.900,106.587,170.1267,13.8281,0.0000
C01452=-42.927,-45.053,106.531,166.9699,12.3897,0.0000
C01453=-43.996,-43.996,106.568,167.3037,12.6959,0.0000
C01454=-45.053,-42.928,106.530,167.6104,13.0302,0.0000
C01455=-46.900,-41.119,106.587,166.1714,9.8715,0.0000
C01456=-50.723,-39.796,107.888,172.6591,-0.7987,0.0000
C01457=-55.853,-42.718,111.064,-178.9427,0.8013,0.0000
C01458=-63.009,-48.291,115.193,-179.1494,0.6513,0.0000
C01459=-71.737,-55.044,119.116,-179.8005,0.1531,0.0000
C01460=-89.648,-11.804,119.116,179.7507,-0.0328,0.0000
C01461=-78.701,-10.407,115.193,178.9381,-0.1410,0.0000
C01462=-69.700,-9.288,111.064,178.6859,-0.1811,0.0000
C01463=-64.006,-7.726,107.888,-174.2350,4.6450,0.0000
C01464=-62.239,-4.087,106.587,-177.0816,16.5478,0.0000
C01465=-62.212,-1.503,106.531,179.5241,17.6914,0.0000
C01466=-62.220,0.000,106.568,179.9997,17.6722,0.0000
C01467=-62.212,1.502,106.530,-179.5239,17.6913,0.0000
C01468=-62.239,4.088,106.587,177.0800,16.5469,0.0000
C01469=-64.006,7.727,107.888,174.2353,4.6444,0.0000
C01470=-69.700,9.288,111.064,-178.6859,-0.1811,0.0000
C01471=-78.701,10.407,115.193,-178.9381,-0.1410,0.0000
C01472=-89.648,11.804,119.116,-179.7507,-0.0328,0.0000
C01473=-71.737,55.044,119.116,179.8005,0.1531,0.0000
C01474=-63.009,48.291,115.193,179.1494,0.6513,0.0000
C01475=-55.853,42.718,111.064,178.9427,0.8013,0.0000
C01476=-50.723,39.796,107.888,-172.6585,-0.7985,0.0000
C01477=-46.900,41.119,106.587,-166.1719,9.8733,0.0000
C01478=-45.053,42.927,106.531,-167.6103,13.0301,0.0000
C01479=-43.996,43.996,106.568,-167.3041,12.6963,0.0000
C01480=-42.928,45.053,106.530,-166.9698,12.3896,0.0000
C01481=-41.119,46.900,106.587,-170.1285,13.8286,0.0000
C01482=-39.796,50.723,107.888,179.2013,7.3409,0.0000
C01483=-42.718,55.853,111.064,-179.1987,-1.0573,0.0000
C01484=-48.291,63.009,115.193,-179.3487,-0.8506,0.0000
C01485=-55.044,71.737,119.116,-179.8469,-0.1995,0.0000
C01486=-11.804,89.648,119.116,179.9672,0.2493,0.0000
C01487=-10.407,78.701,115.193,179.8590,1.0619,0.0000
C01488=-9.288,69.700,111.064,179.8189,1.3141,0.0000
C01489=-7.727,64.006,107.888,-175.3556,-5.7647,0.0000
C01490=-4.088,62.239,106.587,-163.4531,-2.9200,0.0000
C01491=-1.502,62.212,106.530,-162.3087,0.4761,0.0000
C01492=0.000,62.220,106.568,-162.3278,-0.0003,0.0000
C01493=0.000,61.595,108.678,-164.7108,-0.0002,0.0000
C01494=1.446,61.587,108.639,-164.6863,-0.3866,0.0000
C01495=3.992,61.623,108.697,-165.7366,2.5712,0.0000
C01496=7.621,63.469,110.018,-176.1886,4.8019,0.0000
C01497=9.195,69.347,113.234,179.8602,-1.0343,0.0000
C01498=10.356,78.559,117.388,179.9222,-0.5895,0.0000
C01499=48.226,62.872,117.388,-179.6382,0.4718,0.0000
C01500=42.534,55.538,113.234,-179.3675,0.8303,0.0000
C01501=39.491,50.268,110.018,179.2956,-6.0796,0.0000
C01502=40.751,46.396,108.697,-171.5811,-11.9427,0.0000
C01503=42.526,44.571,108.639,-168.7785,-10.6945,0.0000
C01504=43.554,43.554,108.678,-169.0596,-10.9402,0.0000
C01505=44.571,42.527,108.639,-169.3055,-11.2216,0.0000
C01506=46.397,40.751,108.697,-168.0569,-8.4173,0.0000
C01507=50.268,39.491,110.019,-173.9210,0.7045,0.0000
C01508=55.538,42.534,113.234,179.1697,-0.6325,0.0000
C01509=62.872,48.226,117.388,179.5282,-0.3618,0.0000
C01510=78.559,10.356,117.388,-179.4105,0.0778,0.0000
C01511=69.347,9.195,113.234,-178.9657,0.1398,0.0000
C01512=63.469,7.621,110.018,175.1981,-3.8114,0.0000
C01513=61.623,3.992,108.697,177.4288,-14.2634,0.0000
C01514=61.587,1.446,108.639,-179.6134,-15.3137,0.0000
C01515=61.595,0.000,108.678,-179.9998,-15.2892,0.0000
C01516=61.587,-1.445,108.639,179.6133,-15.3137,0.0000
C01517=61.623,-3.992,108.697,-177.4274,-14.2626,0.0000
C01518=63.470,-7.621,110.019,-175.1983,-3.8109,0.0000
C01519=69.347,-9.195,113.234,178.9657,0.1398,0.0000
C01520=78.559,-10.356,117.388,179.4105,0.0778,0.0000
C01521=62.872,-48.226,117.388,-179.5282,-0.3618,0.0000
C01522=55.538,-42.534,113.234,-179.1697,-0.6325,0.0000
C01523=50.268,-39.491,110.018,173.9204,0.7044,0.0000
C01524=46.396,-40.751,108.697,168.0573,-8.4189,0.0000
C01525=44.571,-42.526,108.639,169.3055,-11.2215,0.0000
C01526=43.554,-43.554,108.678,169.0598,-10.9404,0.0000
C01527=42.527,-44.571,108.639,168.7784,-10.6945,0.0000
C01528=40.751,-46.397,108.697,171.5827,-11.9431,0.0000
C01529=39.491,-50.268,110.019,-179.2955,-6.0790,0.0000
C01530=42.534,-55.538,113.234,179.3675,0.8303,0.0000
C01531=48.226,-62.872,117.388,179.6382,0.4718,0.0000
C01532=10.356,-78.559,117.388,-179.9222,-0.5895,0.0000
C01533=9.195,-69.347,113.234,-179.8602,-1.0343,0.0000
C01534=7.621,-63.469,110.018,176.1886,4.8019,0.0000
C01535=3.992,-61.623,108.697,165.7366,2.5712,0.0000
C01536=1.446,-61.587,108.639,164.6863,-0.3866,0.0000
C01537=0.000,-61.595,108.678,164.7108,-0.0002,0.0000
C01538=0.000,-61.595,108.678,164.7108,-0.0002,0.0000
C01539=-1.445,-61.587,108.639,164.6863,0.3867,0.0000
C01540=-3.992,-61.623,108.697,165.7374,-2.5726,0.0000
C01541=-7.621,-63.470,110.019,176.1891,-4.8017,0.0000
C01542=-9.195,-69.347,113.234,-179.8602,1.0343,0.0000
C01543=-10.356,-78.559,117.388,-179.9222,0.5895,0.0000
C01544=-48.226,-62.872,117.388,179.6382,-0.4718,0.0000
C01545=-42.534,-55.538,113.234,179.3675,-0.8303,0.0000
C01546=-39.491,-50.268,110.018,-179.2956,6.0796,0.0000
C01547=-40.751,-46.396,108.697,171.5811,11.9427,0.0000
C01548=-42.526,-44.571,108.639,168.7785,10.6945,0.0000
C01549=-43.554,-43.554,108.678,169.0596,10.9402,0.0000
C01550=-44.571,-42.527,108.639,169.3055,11.2216,0.0000
C01551=-46.397,-40.751,108.697,168.0569,8.4173,0.0000
C01552=-50.268,-39.491,110.019,173.9210,-0.7045,0.0000
C01553=-55.538,-42.534,113.234,-179.1697,0.6325,0.0000
C01554=-62.872,-48.226,117.388,-179.5282,0.3618,0.0000
C01555=-78.559,-10.356,117.388,179.4105,-0.0778,0.0000
C01556=-69.347,-9.195,113.234,178.9657,-0.1398,0.0000
C01557=-63.469,-7.621,110.018,-175.1981,3.8114,0.0000
C01558=-61.623,-3.992,108.697,-177.4288,14.2634,0.0000
C01559=-61.587,-1.446,108.639,179.6134,15.3137,0.0000
C01560=-61.595,0.000,108.678,179.9998,15.2892,0.0000
C01561=-61.587,1.445,108.639,-179.6133,15.3137,0.0000
C01562=-61.623,3.992,108.697,177.4274,14.2626,0.0000
C01563=-63.470,7.621,110.019,175.1983,3.8109,0.0000
C01564=-69.347,9.195,113.234,-178.9657,-0.1398,0.0000
C01565=-78.559,10.356,117.388,-179.4105,-0.0778,0.0000
C01566=-62.872,48.226,117.388,179.5282,0.3618,0.0000
C01567=-55.538,42.534,113.234,179.1697,0.6325,0.0000
C01568=-50.268,39.491,110.018,-173.9204,-0.7044,0.0000
C01569=-46.396,40.751,108.697,-168.0573,8.4189,0.0000
C01570=-44.571,42.526,108.639,-169.3055,11.2215,0.0000
C01571=-43.554,43.554,108.678,-169.0598,10.9404,0.0000
C01572=-42.527,44.571,108.639,-168.7784,10.6945,0.0000
C01573=-40.751,46.397,108.697,-171.5827,11.9431,0.0000
C01574=-39.491,50.268,110.019,179.2955,6.0790,0.0000
C01575=-42.534,55.538,113.234,-179.3675,-0.8303,0.0000
C01576=-48.226,62.872,117.388,-179.6382,-0.4718,0.0000
C01577=-10.356,78.559,117.388,179.9222,0.5895,0.0000
C01578=-9.195,69.347,113.234,179.8602,1.0343,0.0000
C01579=-7.621,63.470,110.019,-176.1891,-4.8017,0.0000
C01580=-3.992,61.623,108.697,-165.7374,-2.5726,0.0000
C01581=-1.445,61.587,108.639,-164.6863,0.3867,0.0000
C01582=0.000,61.595,108.678,-164.7108,-0.0002,0.0000
C01583=0.000,61.062,110.812,-167.2795,-0.0001,0.0000
C01584=1.397,61.054,110.773,-167.2490,-0.3031,0.0000
C01585=3.910,61.097,110.832,-168.1748,2.1705,0.0000
C01586=7.533,63.025,112.171,-177.0134,3.8097,0.0000
C01587=9.126,69.087,115.417,179.9035,-0.7237,0.0000
C01588=10.335,78.500,119.587,179.9875,-0.0950,0.0000
C01589=48.200,62.816,119.587,-179.9417,0.0760,0.0000
C01590=42.399,55.304,115.417,-179.5565,0.5799,0.0000
C01591=39.239,49.892,112.171,179.4159,-4.8004,0.0000
C01592=40.438,45.967,110.832,-173.0868,-9.9177,0.0000
C01593=42.184,44.160,110.773,-170.7001,-8.8821,0.0000
C01594=43.178,43.178,110.812,-170.9309,-9.0689,0.0000
C01595=44.159,42.185,110.773,-171.1179,-9.2999,0.0000
C01596=45.967,40.437,110.832,-170.0820,-6.9118,0.0000
C01597=49.892,39.239,112.171,-175.2001,0.5842,0.0000
C01598=55.304,42.399,115.417,179.4201,-0.4435,0.0000
C01599=62.816,48.200,119.587,179.9240,-0.0583,0.0000
C01600=78.500,10.335,119.587,-179.9050,0.0125,0.0000
C01601=69.087,9.126,115.417,-179.2763,0.0965,0.0000
C01602=63.025,7.533,112.171,176.1903,-2.9866,0.0000
C01603=61.097,3.910,110.832,177.8295,-11.8252,0.0000
C01604=61.054,1.397,110.773,-179.6969,-12.7510,0.0000
C01605=61.062,0.000,110.812,-179.9999,-12.7205,0.0000
C01606=61.054,-1.396,110.773,179.6969,-12.7510,0.0000
C01607=61.097,-3.910,110.832,-177.8283,-11.8245,0.0000
C01608=63.025,-7.533,112.171,-176.1905,-2.9862,0.0000
C01609=69.087,-9.126,115.417,179.2763,0.0965,0.0000
C01610=78.500,-10.335,119.587,179.9050,0.0125,0.0000
C01611=62.816,-48.200,119.587,-179.9240,-0.0583,0.0000
C01612=55.304,-42.399,115.417,-179.4201,-0.4435,0.0000
C01613=49.892,-39.239,112.171,175.1996,0.5841,0.0000
C01614=45.967,-40.438,110.832,170.0823,-6.9132,0.0000
C01615=44.160,-42.184,110.773,171.1179,-9.2999,0.0000
C01616=43.178,-43.178,110.812,170.9311,-9.0691,0.0000
C01617=42.185,-44.159,110.773,170.7001,-8.8821,0.0000
C01618=40.437,-45.967,110.832,173.0882,-9.9180,0.0000
C01619=39.239,-49.892,112.171,-179.4158,-4.7999,0.0000
C01620=42.399,-55.304,115.417,179.5565,0.5799,0.0000
C01621=48.200,-62.816,119.587,179.9417,0.0760,0.0000
C01622=10.335,-78.500,119.587,-179.9875,-0.0950,0.0000
C01623=9.126,-69.087,115.417,-179.9035,-0.7237,0.0000
C01624=7.533,-63.025,112.171,177.0134,3.8097,0.0000
C01625=3.910,-61.097,110.832,168.1748,2.1705,0.0000
C01626=1.397,-61.054,110.773,167.2490,-0.3031,0.0000
C01627=0.000,-61.062,110.812,167.2795,-0.0001,0.0000
C01628=0.000,-61.062,110.812,167.2795,-0.0001,0.0000
C01629=-1.396,-61.054,110.773,167.2490,0.3031,0.0000
C01630=-3.910,-61.097,110.832,168.1755,-2.1717,0.0000
C01631=-7.533,-63.025,112.171,177.0138,-3.8095,0.0000
C01632=-9.126,-69.087,115.417,-179.9035,0.7237,0.0000
C01633=-10.335,-78.500,119.587,-179.9875,0.0950,0.0000
C01634=-48.200,-62.816,119.587,179.9417,-0.0760,0.0000
C01635=-42.399,-55.304,115.417,179.5565,-0.5799,0.0000
C01636=-39.239,-49.892,112.171,-179.4159,4.8004,0.0000
C01637=-40.438,-45.967,110.832,173.0868,9.9177,0.0000
C01638=-42.184,-44.160,110.773,170.7001,8.8821,0.0000
C01639=-43.178,-43.178,110.812,170.9309,9.0689,0.0000
C01640=-44.159,-42.185,110.773,171.1179,9.2999,0.0000
C01641=-45.967,-40.437,110.832,170.0820,6.9118,0.0000
C01642=-49.892,-39.239,112.171,175.2001,-0.5842,0.0000
C01643=-55.304,-42.399,115.417,-179.4201,0.4435,0.0000
C01644=-62.816,-48.200,119.587,-179.9240,0.0583,0.0000
C01645=-78.500,-10.335,119.587,179.9050,-0.0125,0.0000
C01646=-69.087,-9.126,115.417,179.2763,-0.0965,0.0000
C01647=-63.025,-7.533,112.171,-176.1903,2.9866,0.0000
C01648=-61.097,-3.910,110.832,-177.8295,11.8252,0.0000
C01649=-61.054,-1.397,110.773,179.6969,12.7510,0.0000
C01650=-61.062,0.000,110.812,179.9999,12.7205,0.0000
C01651=-61.054,1.396,110.773,-179.6969,12.7510,0.0000
C01652=-61.097,3.910,110.832,177.8283,11.8245,0.0000
C01653=-63.025,7.533,112.171,176.1905,2.9862,0.0000
C01654=-69.087,9.126,115.417,-179.2763,-0.0965,0.0000
C01655=-78.500,10.335,119.587,-179.9050,-0.0125,0.0000
C01656=-62.816,48.200,119.587,179.9240,0.0583,0.0000
C01657=-55.304,42.399,115.417,179.4201,0.4435,0.0000
C01658=-49.892,39.239,112.171,-175.1996,-0.5841,0.0000
C01659=-45.967,40.438,110.832,-170.0823,6.9132,0.0000
C01660=-44.160,42.184,110.773,-171.1179,9.2999,0.0000
C01661=-43.178,43.178,110.812,-170.9311,9.0691,0.0000
C01662=-42.185,44.159,110.773,-170.7001,8.8821,0.0000
C01663=-40.437,45.967,110.832,-173.0882,9.9180,0.0000
C01664=-39.239,49.892,112.171,179.4158,4.7999,0.0000
C01665=-42.399,55.304,115.417,-179.5565,-0.5799,0.0000
C01666=-48.200,62.816,119.587,-179.9417,-0.0760,0.0000
C01667=-10.335,78.500,119.587,179.9875,0.0950,0.0000
C01668=-9.126,69.087,115.417,179.9035,0.7237,0.0000
C01669=-7.533,63.025,112.171,-177.0138,-3.8095,0.0000
C01670=-3.910,61.097,110.832,-168.1755,-2.1717,0.0000
C01671=-1.396,61.054,110.773,-167.2490,0.3031,0.0000
C01672=0.000,61.062,110.812,-167.2795,-0.0001,0.0000
C01673=0.000,60.629,112.969,-170.0330,-0.0001,0.0000
C01674=1.357,60.620,112.930,-169.9958,-0.2252,0.0000
C01675=3.843,60.670,112.989,-170.7655,1.7193,0.0000
C01676=7.465,62.679,114.343,-177.8357,2.7874,0.0000
C01677=9.082,68.923,117.611,179.9488,-0.3874,0.0000
C01678=42.314,55.158,117.611,-179.7623,0.3101,0.0000
C01679=39.042,49.599,114.343,179.5586,-3.4993,0.0000
C01680=40.183,45.618,112.989,-174.6448,-7.7553,0.0000
C01681=41.905,43.825,112.930,-172.7331,-6.9532,0.0000
C01682=42.871,42.871,112.969,-172.9165,-7.0834,0.0000
C01683=43.824,41.906,112.930,-173.0467,-7.2668,0.0000
C01684=45.618,40.182,112.989,-172.2445,-5.3541,0.0000
C01685=49.599,39.042,114.343,-176.5011,0.4415,0.0000
C01686=55.158,42.314,117.611,179.6899,-0.2377,0.0000
C01687=68.923,9.082,117.611,-179.6126,0.0512,0.0000
C01688=62.679,7.465,114.343,177.2126,-2.1643,0.0000
C01689=60.670,3.843,112.989,178.2807,-9.2345,0.0000
C01690=60.620,1.357,112.930,-179.7748,-10.0042,0.0000
C01691=60.629,0.000,112.969,-179.9999,-9.9670,0.0000
C01692=60.620,-1.356,112.930,179.7748,-10.0042,0.0000
C01693=60.670,-3.844,112.989,-178.2798,-9.2339,0.0000
C01694=62.679,-7.465,114.343,-177.2128,-2.1639,0.0000
C01695=68.923,-9.082,117.611,179.6126,0.0512,0.0000
C01696=55.158,-42.314,117.611,-179.6899,-0.2377,0.0000
C01697=49.599,-39.042,114.343,176.5007,0.4414,0.0000
C01698=45.618,-40.183,112.989,172.2447,-5.3552,0.0000
C01699=43.825,-41.905,112.930,173.0468,-7.2669,0.0000
C01700=42.871,-42.871,112.969,172.9166,-7.0835,0.0000
C01701=41.906,-43.824,112.930,172.7332,-6.9533,0.0000
C01702=40.182,-45.618,112.989,174.6459,-7.7555,0.0000
C01703=39.042,-49.599,114.343,-179.5585,-3.4989,0.0000
C01704=42.314,-55.158,117.611,179.7623,0.3101,0.0000
C01705=9.082,-68.923,117.611,-179.9488,-0.3874,0.0000
C01706=7.465,-62.679,114.343,177.8357,2.7874,0.0000
C01707=3.843,-60.670,112.989,170.7655,1.7193,0.0000
C01708=1.357,-60.620,112.930,169.9958,-0.2252,0.0000
C01709=0.000,-60.629,112.969,170.0330,-0.0001,0.0000
C01710=0.000,-60.629,112.969,170.0330,-0.0001,0.0000
C01711=-1.356,-60.620,112.930,169.9958,0.2252,0.0000
C01712=-3.844,-60.670,112.989,170.7661,-1.7202,0.0000
C01713=-7.465,-62.679,114.343,177.8361,-2.7872,0.0000
C01714=-9.082,-68.923,117.611,-179.9488,0.3874,0.0000
C01715=-42.314,-55.158,117.611,179.7623,-0.3101,0.0000
C01716=-39.042,-49.599,114.343,-179.5586,3.4993,0.0000
C01717=-40.183,-45.618,112.989,174.6448,7.7553,0.0000
C01718=-41.905,-43.825,112.930,172.7331,6.9532,0.0000
C01719=-42.871,-42.871,112.969,172.9165,7.0834,0.0000
C01720=-43.824,-41.906,112.930,173.0467,7.2668,0.0000
C01721=-45.618,-40.182,112.989,172.2445,5.3541,0.0000
C01722=-49.599,-39.042,114.343,176.5011,-0.4415,0.0000
C01723=-55.158,-42.314,117.611,-179.6899,0.2377,0.0000
C01724=-68.923,-9.082,117.611,179.6126,-0.0512,0.0000
C01725=-62.679,-7.465,114.343,-177.2126,2.1643,0.0000
C01726=-60.670,-3.843,112.989,-178.2807,9.2345,0.0000
C01727=-60.620,-1.357,112.930,179.7748,10.0042,0.0000
C01728=-60.629,0.000,112.969,179.9999,9.9670,0.0000
C01729=-60.620,1.356,112.930,-179.7748,10.0042,0.0000
C01730=-60.670,3.844,112.989,178.2798,9.2339,0.0000
C01731=-62.679,7.465,114.343,177.2128,2.1639,0.0000
C01732=-68.923,9.082,117.611,-179.6126,-0.0512,0.0000
C01733=-55.158,42.314,117.611,179.6899,0.2377,0.0000
C01734=-49.599,39.042,114.343,-176.5007,-0.4414,0.0000
C01735=-45.618,40.183,112.989,-172.2447,5.3552,0.0000
C01736=-43.825,41.905,112.930,-173.0468,7.2669,0.0000
C01737=-42.871,42.871,112.969,-172.9166,7.0835,0.0000
C01738=-41.906,43.824,112.930,-172.7332,6.9533,0.0000
C01739=-40.182,45.618,112.989,-174.6459,7.7555,0.0000
C01740=-39.042,49.599,114.343,179.5585,3.4989,0.0000
C01741=-42.314,55.158,117.611,-179.7623,-0.3101,0.0000
C01742=-9.082,68.923,117.611,179.9488,0.3874,0.0000
C01743=-7.465,62.679,114.343,-177.8361,-2.7872,0.0000
C01744=-3.844,60.670,112.989,-170.7661,-1.7202,0.0000
C01745=-1.356,60.620,112.930,-169.9958,0.2252,0.0000
C01746=0.000,60.629,112.969,-170.0330,-0.0001,0.0000
C01747=0.000,60.303,115.145,-172.9644,-0.0000,0.0000
C01748=1.327,60.294,115.105,-172.9200,-0.1525,0.0000
C01749=3.793,60.350,115.165,-173.5036,1.2221,0.0000
C01750=7.417,62.439,116.529,-178.6630,1.7334,0.0000
C01751=9.066,68.861,119.810,179.9959,-0.0315,0.0000
C01752=42.282,55.103,119.810,-179.9807,0.0252,0.0000
C01753=38.906,49.396,116.529,179.7195,-2.1706,0.0000
C01754=39.991,45.356,115.165,-176.2562,-5.4612,0.0000
C01755=41.696,43.572,115.105,-174.8740,-4.9120,0.0000
C01756=42.641,42.641,115.145,-175.0125,-4.9874,0.0000
C01757=43.572,41.696,115.105,-175.0879,-5.1260,0.0000
C01758=45.356,39.991,115.165,-174.5388,-3.7430,0.0000
C01759=49.396,38.906,116.529,-177.8297,0.2805,0.0000
C01760=55.103,42.282,119.810,179.9748,-0.0193,0.0000
C01761=68.861,9.066,119.810,-179.9685,0.0041,0.0000
C01762=62.439,7.417,116.529,178.2666,-1.3370,0.0000
C01763=60.350,3.793,115.165,178.7779,-6.4964,0.0000
C01764=60.294,1.327,115.105,-179.8475,-7.0800,0.0000
C01765=60.303,0.000,115.145,-180.0000,-7.0356,0.0000
C01766=60.294,-1.327,115.105,179.8476,-7.0800,0.0000
C01767=60.350,-3.794,115.165,-178.7772,-6.4959,0.0000
C01768=62.440,-7.418,116.529,-178.2668,-1.3368,0.0000
C01769=68.861,-9.066,119.810,179.9685,0.0041,0.0000
C01770=55.103,-42.282,119.810,-179.9748,-0.0193,0.0000
C01771=49.396,-38.906,116.529,177.8294,0.2805,0.0000
C01772=45.356,-39.991,115.165,174.5388,-3.7438,0.0000
C01773=43.572,-41.696,115.105,175.0880,-5.1260,0.0000
C01774=42.641,-42.641,115.145,175.0126,-4.9875,0.0000
C01775=41.696,-43.572,115.105,174.8740,-4.9121,0.0000
C01776=39.991,-45.356,115.165,176.2570,-5.4612,0.0000
C01777=38.906,-49.396,116.529,-179.7195,-2.1703,0.0000
C01778=42.282,-55.103,119.810,179.9807,0.0252,0.0000
C01779=9.066,-68.861,119.810,-179.9959,-0.0315,0.0000
C01780=7.417,-62.439,116.529,178.6630,1.7334,0.0000
C01781=3.793,-60.350,115.165,173.5036,1.2221,0.0000
C01782=1.327,-60.294,115.105,172.9200,-0.1525,0.0000
C01783=0.000,-60.303,115.145,172.9644,-0.0000,0.0000
C01784=0.000,-60.303,115.145,172.9644,-0.0000,0.0000
C01785=-1.327,-60.294,115.105,172.9200,0.1524,0.0000
C01786=-3.794,-60.350,115.165,173.5041,-1.2228,0.0000
C01787=-7.418,-62.440,116.529,178.6632,-1.7332,0.0000
C01788=-9.066,-68.861,119.810,-179.9959,0.0315,0.0000
C01789=-42.282,-55.103,119.810,179.9807,-0.0252,0.0000
C01790=-38.906,-49.396,116.529,-179.7195,2.1706,0.0000
C01791=-39.991,-45.356,115.165,176.2562,5.4612,0.0000
C01792=-41.696,-43.572,115.105,174.8740,4.9120,0.0000
C01793=-42.641,-42.641,115.145,175.0125,4.9874,0.0000
C01794=-43.572,-41.696,115.105,175.0879,5.1260,0.0000
C01795=-45.356,-39.991,115.165,174.5388,3.7430,0.0000
C01796=-49.396,-38.906,116.529,177.8297,-0.2805,0.0000
C01797=-55.103,-42.282,119.810,-179.9748,0.0193,0.0000
C01798=-68.861,-9.066,119.810,179.9685,-0.0041,0.0000
C01799=-62.439,-7.417,116.529,-178.2666,1.3370,0.0000
C01800=-60.350,-3.793,115.165,-178.7779,6.4964,0.0000
C01801=-60.294,-1.327,115.105,179.8475,7.0800,0.0000
C01802=-60.303,0.000,115.145,180.0000,7.0356,0.0000
C01803=-60.294,1.327,115.105,-179.8476,7.0800,0.0000
C01804=-60.350,3.794,115.165,178.7772,6.4959,0.0000
C01805=-62.440,7.418,116.529,178.2668,1.3368,0.0000
C01806=-68.861,9.066,119.810,-179.9685,-0.0041,0.0000
C01807=-55.103,42.282,119.810,179.9748,0.0193,0.0000
C01808=-49.396,38.906,116.529,-177.8294,-0.2805,0.0000
C01809=-45.356,39.991,115.165,-174.5388,3.7438,0.0000
C01810=-43.572,41.696,115.105,-175.0880,5.1260,0.0000
C01811=-42.641,42.641,115.145,-175.0126,4.9875,0.0000
C01812=-41.696,43.572,115.105,-174.8740,4.9121,0.0000
C01813=-39.991,45.356,115.165,-176.2570,5.4612,0.0000
C01814=-38.906,49.396,116.529,179.7195,2.1703,0.0000
C01815=-42.282,55.103,119.810,-179.9807,-0.0252,0.0000
C01816=-9.066,68.861,119.810,179.9959,0.0315,0.0000
C01817=-7.418,62.440,116.529,-178.6632,-1.7332,0.0000
C01818=-3.794,60.350,115.165,-173.5041,-1.2228,0.0000
C01819=-1.327,60.294,115.105,-172.9200,0.1524,0.0000
C01820=0.000,60.303,115.145,-172.9644,-0.0000,0.0000
C01821=0.000,60.092,117.335,-176.0598,-0.0000,0.0000
C01822=1.308,60.081,117.295,-176.0080,-0.0834,0.0000
C01823=3.761,60.142,117.355,-176.3792,0.6856,0.0000
C01824=7.392,62.312,118.725,-179.5035,0.6460,0.0000
C01825=38.834,49.289,118.725,179.8943,-0.8078,0.0000
C01826=39.867,45.187,117.355,-177.9220,-3.0457,0.0000
C01827=41.559,43.408,117.295,-177.1161,-2.7662,0.0000
C01828=42.492,42.492,117.335,-177.2117,-2.7883,0.0000
C01829=43.408,41.560,117.295,-177.2337,-2.8839,0.0000
C01830=45.187,39.867,117.355,-176.9544,-2.0775,0.0000
C01831=49.289,38.834,118.726,-179.1923,0.1057,0.0000
C01832=62.312,7.392,118.725,179.3540,-0.4965,0.0000
C01833=60.142,3.761,117.355,179.3144,-3.6208,0.0000
C01834=60.081,1.308,117.295,-179.9166,-3.9920,0.0000
C01835=60.092,0.000,117.335,-180.0000,-3.9402,0.0000
C01836=60.081,-1.307,117.295,179.9167,-3.9920,0.0000
C01837=60.142,-3.762,117.355,-179.3140,-3.6204,0.0000
C01838=62.312,-7.392,118.726,-179.3541,-0.4964,0.0000
C01839=49.289,-38.834,118.725,179.1922,0.1057,0.0000
C01840=45.187,-39.867,117.355,176.9543,-2.0780,0.0000
C01841=43.408,-41.559,117.295,177.2338,-2.8839,0.0000
C01842=42.492,-42.492,117.335,177.2117,-2.7883,0.0000
C01843=41.560,-43.408,117.295,177.1161,-2.7663,0.0000
